EC00432=28.1117,15118.3294
EC00433=28.1001,15120.0000
EC00434=28.1117,15121.6706
EC00435=26.6025,15124.1349
EC00436=8.4383,15127.1678
EC00437=-0.0548,15127.9465
EC00438=-0.0188,15127.8844
EC00439=-0.0094,15127.7630
EC00440=-0.0057,15127.6803
EC00441=-0.5045,15127.7585
EC00442=-1.1939,15129.4604
EC00443=-0.7971,15132.4636
EC00444=-0.0543,15136.2505
EC00445=-0.0054,15140.3860
EC00446=-0.0052,15144.6140
EC00447=-0.0540,15148.7498
EC00448=-0.7993,15152.5363
EC00449=-1.1940,15155.5394
EC00450=-0.5081,15157.2413
EC00451=-0.0087,15157.3191
EC00452=-0.0113,15157.2369
EC00453=-0.0208,15157.1159
EC00454=-0.0563,15157.0536
EC00455=8.4405,15157.8325
EC00456=26.5997,15160.8660
EC00457=28.1098,15163.3290
EC00458=28.0967,15165.0000
EC00459=28.1098,15166.6710
EC00460=26.5997,15169.1340
EC00461=8.4405,15172.1675
EC00462=-0.0563,15172.9464
EC00463=-0.0208,15172.8841
EC00464=-0.0113,15172.7631
EC00465=-0.0087,15172.6809
EC00466=-0.5081,15172.7587
EC00467=-1.1940,15174.4606
EC00468=-0.7993,15177.4637
EC00469=-0.0540,15181.2502
EC00470=-0.0052,15185.3860
EC00471=-0.0054,15189.6140
EC00472=-0.0543,15193.7495
EC00473=-0.7971,15197.5364
EC00474=-1.1939,15200.5396
EC00475=-0.5045,15202.2415
EC00476=-0.0057,15202.3197
EC00477=-0.0094,15202.2370
EC00478=-0.0188,15202.1156
EC00479=-0.0548,15202.0535
EC00480=8.4383,15202.8322
EC00481=26.6025,15205.8651
EC00482=28.1117,15208.3294
EC00483=28.1001,15210.0000
EC00484=26.2576,15210.0000
EC00485=26.2720,15211.6025
EC00486=24.7331,15214.0449
EC00487=7.3770,15217.0981
EC00488=-0.0435,15217.8538
EC00489=-0.0134,15217.7815
EC00490=-0.0020,15217.6711
EC00491=-0.0031,15217.6022
EC00492=-0.3615,15217.6844
EC00493=-0.8397,15219.3971
EC00494=-0.5442,15222.4165
EC00495=-0.0362,15226.2223
EC00496=-0.0054,15230.3773
EC00497=-0.0052,15234.6227
EC00498=-0.0384,15238.7775
EC00499=-0.5441,15242.5833
EC00500=-0.8412,15245.6027
EC00501=-0.3666,15247.3159
EC00502=-0.0016,15247.3980
EC00503=-0.0027,15247.3291
EC00504=-0.0129,15247.2193
EC00505=-0.0389,15247.1468
EC00506=7.3773,15247.9017
EC00507=24.7330,15250.9551
EC00508=26.2704,15253.3970
EC00509=26.2558,15255.0000
EC00510=26.2704,15256.6030
EC00511=24.7330,15259.0449
EC00512=7.3727,15262.0983
EC00513=-0.0389,15262.8532
EC00514=-0.0129,15262.7807
EC00515=-0.0027,15262.6709
EC00516=-0.0016,15262.6020
EC00517=-0.3666,15262.6841
EC00518=-0.8412,15264.3973
EC00519=-0.5441,15267.4167
EC00520=-0.0384,15271.2225
EC00521=-0.0052,15275.3773
EC00522=-0.0054,15279.6227
EC00523=-0.0362,15283.7777
EC00524=-0.5442,15287.5835
EC00525=-0.8397,15290.6029
EC00526=-0.3615,15292.3156
EC00527=-0.0031,15292.3978
EC00528=-0.0020,15292.3289
EC00529=-0.0134,15292.2185
EC00530=-0.0435,15292.1462
EC00531=7.3770,15292.9019
EC00532=24.7331,15295.9551
EC00533=26.2720,15298.3975
EC00534=26.2576,15300.0000
EC00535=26.2720,15301.6025
EC00536=24.7327,15304.0449
EC00537=7.3770,15307.0981
EC00538=-0.0435,15307.8538
EC00539=-0.0134,15307.7815
EC00540=-0.0020,15307.6711
EC00541=-0.0031,15307.6022
EC00542=-0.3615,15307.6844
EC00543=-0.8397,15309.3971
EC00544=-0.5442,15312.4165
EC00545=-0.0362,15316.2223
EC00546=-0.0054,15320.3773
EC00547=-0.0052,15324.6227
EC00548=-0.0384,15328.7775
EC00549=-0.5441,15332.5833
EC00550=-0.8412,15335.6027
EC00551=-0.3666,15337.3159
EC00552=-0.0016,15337.3980
EC00553=-0.0027,15337.3291
EC00554=-0.0129,15337.2193
EC00555=-0.0389,15337.1468
EC00556=7.3773,15337.9017
EC00557=24.7330,15340.9551
EC00558=26.2704,15343.3970
EC00559=26.2558,15345.0000
EC00560=26.2704,15346.6030
EC00561=24.7330,15349.0449
EC00562=7.3727,15352.0983
EC00563=-0.0389,15352.8532
EC00564=-0.0129,15352.7807
EC00565=-0.0027,15352.6709
EC00566=-0.0016,15352.6020
EC00567=-0.3666,15352.6841
EC00568=-0.8412,15354.3973
EC00569=-0.5441,15357.4167
EC00570=-0.0384,15361.2225
EC00571=-0.0052,15365.3773
EC00572=-0.0054,15369.6227
EC00573=-0.0362,15373.7777
EC00574=-0.5442,15377.5835
EC00575=-0.8397,15380.6029
EC00576=-0.3615,15382.3156
EC00577=-0.0031,15382.3978
EC00578=-0.0020,15382.3289
EC00579=-0.0134,15382.2185
EC00580=-0.0435,15382.1462
EC00581=7.3770,15382.9019
EC00582=24.7331,15385.9551
EC00583=26.2720,15388.3975
EC00584=26.2576,15390.0000
EC00585=26.2576,15390.0000
EC00586=26.2720,15391.6025
EC00587=24.7327,15394.0449
EC00588=7.3770,15397.0981
EC00589=-0.0435,15397.8538
EC00590=-0.0134,15397.7815
EC00591=-0.0020,15397.6711
EC00592=-0.0031,15397.6022
EC00593=-0.3615,15397.6844
EC00594=-0.8397,15399.3971
EC00595=-0.5442,15402.4165
EC00596=-0.0362,15406.2223
EC00597=-0.0054,15410.3773
EC00598=-0.0052,15414.6227
EC00599=-0.0384,15418.7775
EC00600=-0.5441,15422.5833
EC00601=-0.8412,15425.6027
EC00602=-0.3666,15427.3159
EC00603=-0.0016,15427.3980
EC00604=-0.0027,15427.3291
EC00605=-0.0129,15427.2193
EC00606=-0.0389,15427.1468
EC00607=7.3773,15427.9017
EC00608=24.7330,15430.9551
EC00609=26.2704,15433.3970
EC00610=26.2558,15435.0000
EC00611=26.2704,15436.6030
EC00612=24.7330,15439.0449
EC00613=7.3727,15442.0983
EC00614=-0.0389,15442.8532
EC00615=-0.0129,15442.7807
EC00616=-0.0027,15442.6709
EC00617=-0.0016,15442.6020
EC00618=-0.3666,15442.6841
EC00619=-0.8412,15444.3973
EC00620=-0.5441,15447.4167
EC00621=-0.0384,15451.2225
EC00622=-0.0052,15455.3773
EC00623=-0.0054,15459.6227
EC00624=-0.0362,15463.7777
EC00625=-0.5442,15467.5835
EC00626=-0.8397,15470.6029
EC00627=-0.3615,15472.3156
EC00628=-0.0031,15472.3978
EC00629=-0.0020,15472.3289
EC00630=-0.0134,15472.2185
EC00631=-0.0435,15472.1462
EC00632=7.3770,15472.9019
EC00633=24.7331,15475.9551
EC00634=26.2720,15478.3975
EC00635=26.2576,15480.0000
EC00636=26.2720,15481.6025
EC00637=24.7327,15484.0449
EC00638=7.3770,15487.0981
EC00639=-0.0435,15487.8538
EC00640=-0.0134,15487.7815
EC00641=-0.0020,15487.6711
EC00642=-0.0031,15487.6022
EC00643=-0.3615,15487.6844
EC00644=-0.8397,15489.3971
EC00645=-0.5442,15492.4165
EC00646=-0.0362,15496.2223
EC00647=-0.0054,15500.3773
EC00648=-0.0052,15504.6227
EC00649=-0.0384,15508.7775
EC00650=-0.5441,15512.5833
EC00651=-0.8412,15515.6027
EC00652=-0.3666,15517.3159
EC00653=-0.0016,15517.3980
EC00654=-0.0027,15517.3291
EC00655=-0.0129,15517.2193
EC00656=-0.0389,15517.1468
EC00657=7.3773,15517.9017
EC00658=24.7330,15520.9551
EC00659=26.2704,15523.3970
EC00660=26.2558,15525.0000
EC00661=26.2704,15526.6030
EC00662=24.7330,15529.0449
EC00663=7.3727,15532.0983
EC00664=-0.0389,15532.8532
EC00665=-0.0129,15532.7807
EC00666=-0.0027,15532.6709
EC00667=-0.0016,15532.6020
EC00668=-0.3666,15532.6841
EC00669=-0.8412,15534.3973
EC00670=-0.5441,15537.4167
EC00671=-0.0384,15541.2225
EC00672=-0.0052,15545.3773
EC00673=-0.0054,15549.6227
EC00674=-0.0362,15553.7777
EC00675=-0.5442,15557.5835
EC00676=-0.8397,15560.6029
EC00677=-0.3615,15562.3156
EC00678=-0.0031,15562.3978
EC00679=-0.0020,15562.3289
EC00680=-0.0134,15562.2185
EC00681=-0.0435,15562.1462
EC00682=7.3770,15562.9019
EC00683=24.7327,15565.9551
EC00684=26.2720,15568.3975
EC00685=26.2576,15570.0000
EC00686=24.1993,15570.0000
EC00687=24.2117,15571.5376
EC00688=22.6760,15573.9586
EC00689=6.3608,15577.0327
EC00690=-0.0296,15577.7683
EC00691=-0.0072,15577.6919
EC00692=0.0012,15577.5966
EC00693=0.0004,15577.5446
EC00694=-0.2180,15577.6343
EC00695=-0.4664,15579.3569
EC00696=-0.2743,15582.3884
EC00697=-0.0181,15586.2065
EC00698=-0.0000,15590.3718
EC00699=-0.0000,15594.6278
EC00700=-0.0128,15598.7938
EC00701=-0.2776,15602.6119
EC00702=-0.4673,15605.6434
EC00703=-0.2176,15607.3659
EC00704=0.0009,15607.4553
EC00705=-0.0015,15607.4027
EC00706=-0.0071,15607.3085
EC00707=-0.0275,15607.2322
EC00708=6.3616,15607.9674
EC00709=22.6775,15611.0417
EC00710=24.2122,15613.4634
EC00711=24.1961,15615.0000
EC00712=24.2160,15616.5366
EC00713=22.6769,15618.9583
EC00714=6.3616,15622.0326
EC00715=-0.0275,15622.7678
EC00716=-0.0071,15622.6915
EC00717=-0.0015,15622.5973
EC00718=0.0009,15622.5447
EC00719=-0.2176,15622.6341
EC00720=-0.4673,15624.3566
EC00721=-0.2776,15627.3881
EC00722=-0.0128,15631.2062
EC00723=-0.0000,15635.3722
EC00724=-0.0000,15639.6282
EC00725=-0.0181,15643.7935
EC00726=-0.2743,15647.6116
EC00727=-0.4664,15650.6431
EC00728=-0.2180,15652.3657
EC00729=0.0004,15652.4554
EC00730=0.0012,15652.4034
EC00731=-0.0072,15652.3081
EC00732=-0.0296,15652.2317
EC00733=6.3608,15652.9673
EC00734=22.6760,15656.0414
EC00735=24.2117,15658.4624
EC00736=24.1993,15660.0000
EC00737=24.2117,15661.5365
EC00738=22.6760,15663.9586
EC00739=6.3608,15667.0327
EC00740=-0.0296,15667.7683
EC00741=-0.0072,15667.6919
EC00742=0.0012,15667.5966
EC00743=0.0004,15667.5446
EC00744=-0.2180,15667.6343
EC00745=-0.4664,15669.3569
EC00746=-0.2743,15672.3884
EC00747=-0.0181,15676.2065
EC00748=-0.0000,15680.3718
EC00749=-0.0000,15684.6278
EC00750=-0.0128,15688.7938
EC00751=-0.2776,15692.6119
EC00752=-0.4673,15695.6434
EC00753=-0.2176,15697.3659
EC00754=0.0009,15697.4553
EC00755=-0.0015,15697.4027
EC00756=-0.0071,15697.3085
EC00757=-0.0275,15697.2322
EC00758=6.3616,15697.9674
EC00759=22.6775,15701.0417
EC00760=24.2122,15703.4634
EC00761=24.1961,15705.0000
EC00762=24.2160,15706.5366
EC00763=22.6769,15708.9583
EC00764=6.3616,15712.0326
EC00765=-0.0275,15712.7678
EC00766=-0.0071,15712.6915
EC00767=-0.0015,15712.5973
EC00768=0.0009,15712.5447
EC00769=-0.2176,15712.6341
EC00770=-0.4673,15714.3566
EC00771=-0.2776,15717.3881
EC00772=-0.0128,15721.2062
EC00773=-0.0000,15725.3722
EC00774=-0.0000,15729.6282
EC00775=-0.0181,15733.7935
EC00776=-0.2743,15737.6116
EC00777=-0.4664,15740.6431
EC00778=-0.2180,15742.3657
EC00779=0.0004,15742.4554
EC00780=0.0012,15742.4034
EC00781=-0.0072,15742.3081
EC00782=-0.0296,15742.2317
EC00783=6.3608,15742.9673
EC00784=22.6760,15746.0414
EC00785=24.2117,15748.4624
EC00786=24.1993,15750.0000
EC00787=24.1993,15750.0000
EC00788=24.2117,15751.5365
EC00789=22.6760,15753.9586
EC00790=6.3608,15757.0327
EC00791=-0.0296,15757.7683
EC00792=-0.0072,15757.6919
EC00793=0.0012,15757.5966
EC00794=0.0004,15757.5446
EC00795=-0.2180,15757.6343
EC00796=-0.4664,15759.3569
EC00797=-0.2743,15762.3884
EC00798=-0.0181,15766.2065
EC00799=-0.0000,15770.3718
EC00800=-0.0000,15774.6278
EC00801=-0.0128,15778.7938
EC00802=-0.2776,15782.6119
EC00803=-0.4673,15785.6434
EC00804=-0.2176,15787.3659
EC00805=0.0009,15787.4553
EC00806=-0.0015,15787.4027
EC00807=-0.0071,15787.3085
EC00808=-0.0275,15787.2322
EC00809=6.3616,15787.9674
EC00810=22.6775,15791.0417
EC00811=24.2122,15793.4634
EC00812=24.1961,15795.0000
EC00813=24.2160,15796.5366
EC00814=22.6769,15798.9583
EC00815=6.3616,15802.0326
EC00816=-0.0275,15802.7678
EC00817=-0.0071,15802.6915
EC00818=-0.0015,15802.5973
EC00819=0.0009,15802.5447
EC00820=-0.2176,15802.6341
EC00821=-0.4673,15804.3566
EC00822=-0.2776,15807.3881
EC00823=-0.0128,15811.2062
EC00824=-0.0000,15815.3722
EC00825=-0.0000,15819.6282
EC00826=-0.0181,15823.7935
EC00827=-0.2743,15827.6116
EC00828=-0.4664,15830.6431
EC00829=-0.2180,15832.3657
EC00830=0.0004,15832.4554
EC00831=0.0012,15832.4034
EC00832=-0.0072,15832.3081
EC00833=-0.0296,15832.2317
EC00834=6.3608,15832.9673
EC00835=22.6760,15836.0414
EC00836=24.2117,15838.4624
EC00837=24.1993,15840.0000
EC00838=24.2117,15841.5365
EC00839=22.6760,15843.9586
EC00840=6.3608,15847.0327
EC00841=-0.0296,15847.7683
EC00842=-0.0072,15847.6919
EC00843=0.0012,15847.5966
EC00844=0.0004,15847.5446
EC00845=-0.2180,15847.6343
EC00846=-0.4664,15849.3569
EC00847=-0.2743,15852.3884
EC00848=-0.0181,15856.2065
EC00849=-0.0000,15860.3718
EC00850=-0.0000,15864.6278
EC00851=-0.0128,15868.7938
EC00852=-0.2776,15872.6119
EC00853=-0.4673,15875.6434
EC00854=-0.2176,15877.3659
EC00855=0.0009,15877.4553
EC00856=-0.0015,15877.4027
EC00857=-0.0071,15877.3085
EC00858=-0.0275,15877.2322
EC00859=6.3616,15877.9674
EC00860=22.6775,15881.0417
EC00861=24.2122,15883.4634
EC00862=24.1961,15885.0000
EC00863=24.2160,15886.5366
EC00864=22.6769,15888.9583
EC00865=6.3616,15892.0326
EC00866=-0.0275,15892.7678
EC00867=-0.0071,15892.6915
EC00868=-0.0015,15892.5973
EC00869=0.0009,15892.5447
EC00870=-0.2176,15892.6341
EC00871=-0.4673,15894.3566
EC00872=-0.2776,15897.3881
EC00873=-0.0128,15901.2062
EC00874=-0.0000,15905.3722
EC00875=-0.0000,15909.6282
EC00876=-0.0181,15913.7935
EC00877=-0.2743,15917.6116
EC00878=-0.4664,15920.6431
EC00879=-0.2180,15922.3657
EC00880=0.0004,15922.4554
EC00881=0.0012,15922.4034
EC00882=-0.0072,15922.3081
EC00883=-0.0296,15922.2317
EC00884=6.3608,15922.9673
EC00885=22.6760,15926.0414
EC00886=24.2117,15928.4635
EC00887=24.1993,15930.0000
EC00888=21.8993,15930.0000
EC00889=21.9171,15931.4747
EC00890=20.4142,15933.8756
EC00891=5.3944,15936.9699
EC00892=-0.0194,15937.6906
EC00893=-0.0061,15937.6170
EC00894=0.0006,15937.5429
EC00895=-0.0001,15937.5106
EC00896=-0.0677,15937.6094
EC00897=-0.0727,15939.3401
EC00898=-0.0715,15965.6602
EC00899=-0.0690,15967.3910
EC00900=-0.0010,15967.4898
EC00901=-0.0010,15967.4572
EC00902=-0.0014,15967.3834
EC00903=-0.0171,15967.3085
EC00904=5.3944,15968.0296
EC00905=20.4131,15971.1238
EC00906=21.9192,15973.5256
EC00907=21.8955,15975.0000
EC00908=21.9192,15976.4744
EC00909=20.4131,15978.8762
EC00910=5.3909,15981.9704
EC00911=-0.0171,15982.6915
EC00912=-0.0014,15982.6166
EC00913=-0.0010,15982.5428
EC00914=-0.0010,15982.5102
EC00915=-0.0690,15982.6090
EC00916=-0.0715,15984.3398
EC00917=-0.0727,16010.6599
EC00918=-0.0677,16012.3906
EC00919=-0.0001,16012.4894
EC00920=0.0006,16012.4571
EC00921=-0.0061,16012.3830
EC00922=-0.0194,16012.3094
EC00923=5.3944,16013.0301
EC00924=20.4142,16016.1244
EC00925=21.9171,16018.5253
EC00926=21.8993,16020.0000
EC00927=21.9171,16021.4736
EC00928=20.4141,16023.8767
EC00929=5.3944,16026.9699
EC00930=-0.0194,16027.6906
EC00931=-0.0061,16027.6170
EC00932=0.0006,16027.5429
EC00933=-0.0001,16027.5106
EC00934=-0.0677,16027.6094
EC00935=-0.0727,16029.3401
EC00936=-0.0715,16055.6602
EC00937=-0.0690,16057.3910
EC00938=-0.0010,16057.4898
EC00939=-0.0010,16057.4572
EC00940=-0.0014,16057.3834
EC00941=-0.0171,16057.3085
EC00942=5.3944,16058.0296
EC00943=20.4131,16061.1238
EC00944=21.9192,16063.5256
EC00945=21.8955,16065.0000
EC00946=21.9192,16066.4744
EC00947=20.4131,16068.8762
EC00948=5.3909,16071.9704
EC00949=-0.0171,16072.6915
EC00950=-0.0014,16072.6166
EC00951=-0.0010,16072.5428
EC00952=-0.0010,16072.5102
EC00953=-0.0690,16072.6090
EC00954=-0.0715,16074.3398
EC00955=-0.0727,16100.6599
EC00956=-0.0677,16102.3906
EC00957=-0.0001,16102.4894
EC00958=0.0006,16102.4571
EC00959=-0.0061,16102.3830
EC00960=-0.0194,16102.3094
EC00961=5.3944,16103.0301
EC00962=20.4142,16106.1244
EC00963=21.9171,16108.5253
EC00964=21.8993,16110.0000
EC00965=21.8993,16110.0000
EC00966=21.9171,16111.4736
EC00967=20.4141,16113.8767
EC00968=5.3944,16116.9699
EC00969=-0.0194,16117.6906
EC00970=-0.0061,16117.6170
EC00971=0.0006,16117.5429
EC00972=-0.0001,16117.5106
EC00973=-0.0677,16117.6094
EC00974=-0.0727,16119.3401
EC00975=-0.0715,16145.6602
EC00976=-0.0690,16147.3910
EC00977=-0.0010,16147.4898
EC00978=-0.0010,16147.4572
EC00979=-0.0014,16147.3834
EC00980=-0.0171,16147.3085
EC00981=5.3944,16148.0296
EC00982=20.4131,16151.1238
EC00983=21.9192,16153.5256
EC00984=21.8955,16155.0000
EC00985=21.9192,16156.4744
EC00986=20.4131,16158.8762
EC00987=5.3909,16161.9704
EC00988=-0.0171,16162.6915
EC00989=-0.0014,16162.6166
EC00990=-0.0010,16162.5428
EC00991=-0.0010,16162.5102
EC00992=-0.0690,16162.6090
EC00993=-0.0715,16164.3398
EC00994=-0.0727,16190.6599
EC00995=-0.0677,16192.3906
EC00996=-0.0001,16192.4894
EC00997=0.0006,16192.4571
EC00998=-0.0061,16192.3830
EC00999=-0.0194,16192.3094
EC01000=5.3944,16193.0301
EC01001=20.4142,16196.1244
EC01002=21.9171,16198.5253
EC01003=21.8993,16200.0000
EC01004=21.9171,16201.4736
EC01005=20.4141,16203.8767
EC01006=5.3944,16206.9699
EC01007=-0.0194,16207.6906
EC01008=-0.0061,16207.6170
EC01009=0.0006,16207.5429
EC01010=-0.0001,16207.5106
EC01011=-0.0677,16207.6094
EC01012=-0.0727,16209.3401
EC01013=-0.0715,16235.6602
EC01014=-0.0690,16237.3910
EC01015=-0.0010,16237.4898
EC01016=-0.0010,16237.4572
EC01017=-0.0014,16237.3834
EC01018=-0.0171,16237.3085
EC01019=5.3944,16238.0296
EC01020=20.4131,16241.1238
EC01021=21.9192,16243.5256
EC01022=21.8955,16245.0000
EC01023=21.9192,16246.4744
EC01024=20.4131,16248.8762
EC01025=5.3909,16251.9704
EC01026=-0.0171,16252.6915
EC01027=-0.0014,16252.6166
EC01028=-0.0010,16252.5428
EC01029=-0.0010,16252.5102
EC01030=-0.0690,16252.6090
EC01031=-0.0715,16254.3398
EC01032=-0.0727,16280.6599
EC01033=-0.0677,16282.3906
EC01034=-0.0001,16282.4894
EC01035=0.0006,16282.4571
EC01036=-0.0061,16282.3830
EC01037=-0.0194,16282.3094
EC01038=5.3944,16283.0301
EC01039=20.4141,16286.1233
EC01040=21.9171,16288.5264
EC01041=21.8993,16290.0000
EC01042=19.3355,16290.0000
EC01043=19.3601,16291.4165
EC01044=17.9316,16293.7994
EC01045=4.4629,16296.9134
EC01046=-0.0109,16297.6249
EC01047=-0.0035,16297.5584
EC01048=0.0012,16297.5104
EC01049=-0.0008,16327.4901
EC01050=-0.0004,16327.4412
EC01051=-0.0099,16327.3752
EC01052=4.4644,16328.0867
EC01053=17.9314,16331.2006
EC01054=19.3612,16333.5844
EC01055=19.3375,16335.0000
EC01056=19.3612,16336.4156
EC01057=17.9313,16338.8001
EC01058=4.4644,16341.9133
EC01059=-0.0099,16342.6248
EC01060=-0.0004,16342.5588
EC01061=-0.0008,16342.5099
EC01062=0.0012,16372.4896
EC01063=-0.0035,16372.4416
EC01064=-0.0109,16372.3751
EC01065=4.4629,16373.0866
EC01066=17.9316,16376.2006
EC01067=19.3601,16378.5835
EC01068=19.3355,16380.0000
EC01069=19.3601,16381.4153
EC01070=17.9315,16383.8005
EC01071=4.4629,16386.9134
EC01072=-0.0109,16387.6249
EC01073=-0.0035,16387.5584
EC01074=0.0012,16387.5104
EC01075=-0.0008,16417.4901
EC01076=-0.0004,16417.4412
EC01077=-0.0099,16417.3752
EC01078=4.4644,16418.0867
EC01079=17.9314,16421.2006
EC01080=19.3612,16423.5844
EC01081=19.3375,16425.0000
EC01082=19.3612,16426.4156
EC01083=17.9313,16428.8001
EC01084=4.4644,16431.9133
EC01085=-0.0099,16432.6248
EC01086=-0.0004,16432.5588
EC01087=-0.0008,16432.5099
EC01088=0.0012,16462.4896
EC01089=-0.0035,16462.4416
EC01090=-0.0109,16462.3751
EC01091=4.4629,16463.0866
EC01092=17.9316,16466.2006
EC01093=19.3601,16468.5835
EC01094=19.3355,16470.0000
EC01095=19.3355,16470.0000
EC01096=19.3601,16471.4153
EC01097=17.9315,16473.8005
EC01098=4.4629,16476.9134
EC01099=-0.0109,16477.6249
EC01100=-0.0035,16477.5584
EC01101=0.0012,16477.5104
EC01102=-0.0008,16507.4901
EC01103=-0.0004,16507.4412
EC01104=-0.0099,16507.3752
EC01105=4.4644,16508.0867
EC01106=17.9314,16511.2006
EC01107=19.3612,16513.5844
EC01108=19.3375,16515.0000
EC01109=19.3612,16516.4156
EC01110=17.9313,16518.8001
EC01111=4.4644,16521.9133
EC01112=-0.0099,16522.6248
EC01113=-0.0004,16522.5588
EC01114=-0.0008,16522.5099
EC01115=0.0012,16552.4896
EC01116=-0.0035,16552.4416
EC01117=-0.0109,16552.3751
EC01118=4.4629,16553.0866
EC01119=17.9316,16556.2006
EC01120=19.3601,16558.5835
EC01121=19.3355,16560.0000
EC01122=19.3601,16561.4153
EC01123=17.9315,16563.8005
EC01124=4.4629,16566.9134
EC01125=-0.0109,16567.6249
EC01126=-0.0035,16567.5584
EC01127=0.0012,16567.5104
EC01128=-0.0008,16597.4901
EC01129=-0.0004,16597.4412
EC01130=-0.0099,16597.3752
EC01131=4.4644,16598.0867
EC01132=17.9314,16601.2006
EC01133=19.3612,16603.5844
EC01134=19.3375,16605.0000
EC01135=19.3612,16606.4156
EC01136=17.9313,16608.8001
EC01137=4.4644,16611.9133
EC01138=-0.0099,16612.6248
EC01139=-0.0004,16612.5588
EC01140=-0.0008,16612.5099
EC01141=0.0012,16642.4896
EC01142=-0.0035,16642.4416
EC01143=-0.0109,16642.3751
EC01144=4.4629,16643.0866
EC01145=17.9315,16646.1995
EC01146=19.3601,16648.5847
EC01147=19.3355,16650.0000
EC01148=16.4995,16650.0000
EC01149=16.5281,16651.3641
EC01150=15.2268,16653.7307
EC01151=3.5661,16656.8641
EC01152=-0.0035,16657.5707
EC01153=0.0008,16657.5193
EC01154=0.0002,16687.4799
EC01155=-0.0013,16687.4296
EC01156=3.5658,16688.1360
EC01157=15.2245,16691.2692
EC01158=16.5280,16693.6362
EC01159=16.5019,16695.0000
EC01160=16.5280,16696.3630
EC01161=15.2245,16698.7308
EC01162=3.5623,16701.8640
EC01163=-0.0013,16702.5704
EC01164=0.0002,16702.5201
EC01165=0.0008,16732.4807
EC01166=-0.0035,16732.4293
EC01167=3.5661,16733.1359
EC01168=15.2268,16736.2693
EC01169=16.5281,16738.6359
EC01170=16.4995,16740.0000
EC01171=16.5281,16741.3630
EC01172=15.2212,16743.7318
EC01173=3.5661,16746.8641
EC01174=-0.0035,16747.5707
EC01175=0.0008,16747.5193
EC01176=0.0002,16777.4799
EC01177=-0.0013,16777.4296
EC01178=3.5658,16778.1360
EC01179=15.2245,16781.2692
EC01180=16.5280,16783.6362
EC01181=16.5019,16785.0000
EC01182=16.5280,16786.3630
EC01183=15.2245,16788.7308
EC01184=3.5623,16791.8640
EC01185=-0.0013,16792.5704
EC01186=0.0002,16792.5201
EC01187=0.0008,16822.4807
EC01188=-0.0035,16822.4293
EC01189=3.5661,16823.1359
EC01190=15.2268,16826.2693
EC01191=16.5281,16828.6359
EC01192=16.4995,16830.0000
EC01193=16.4995,16830.0000
EC01194=16.5281,16831.3630
EC01195=15.2212,16833.7318
EC01196=3.5661,16836.8641
EC01197=-0.0035,16837.5707
EC01198=0.0008,16837.5193
EC01199=0.0002,16867.4799
EC01200=-0.0013,16867.4296
EC01201=3.5658,16868.1360
EC01202=15.2245,16871.2692
EC01203=16.5280,16873.6362
EC01204=16.5019,16875.0000
EC01205=16.5280,16876.3630
EC01206=15.2245,16878.7308
EC01207=3.5623,16881.8640
EC01208=-0.0013,16882.5704
EC01209=0.0002,16882.5201
EC01210=0.0008,16912.4807
EC01211=-0.0035,16912.4293
EC01212=3.5661,16913.1359
EC01213=15.2268,16916.2693
EC01214=16.5281,16918.6359
EC01215=16.4995,16920.0000
EC01216=16.5281,16921.3630
EC01217=15.2212,16923.7318
EC01218=3.5661,16926.8641
EC01219=-0.0035,16927.5707
EC01220=0.0008,16927.5193
EC01221=0.0002,16957.4799
EC01222=-0.0013,16957.4296
EC01223=3.5658,16958.1360
EC01224=15.2245,16961.2692
EC01225=16.5280,16963.6362
EC01226=16.5019,16965.0000
EC01227=16.5280,16966.3630
EC01228=15.2245,16968.7308
EC01229=3.5623,16971.8640
EC01230=-0.0013,16972.5704
EC01231=0.0002,16972.5201
EC01232=0.0008,17002.4807
EC01233=-0.0035,17002.4293
EC01234=3.5661,17003.1359
EC01235=15.2212,17006.2682
EC01236=16.5281,17008.6370
EC01237=16.4995,17010.0000
EC01238=13.3790,17010.0000
EC01239=13.4131,17011.3191
EC01240=12.2840,17013.6720
EC01241=2.6850,17016.8225
EC01242=-0.0028,17017.5303
EC01243=0.0000,17017.5014
EC01244=0.0010,17047.4983
EC01245=0.0007,17047.4688
EC01246=2.6894,17048.1772
EC01247=12.2833,17051.3279
EC01248=13.4108,17053.6816
EC01249=13.3770,17055.0000
EC01250=13.4108,17056.3184
EC01251=12.2833,17058.6728
EC01252=2.6858,17061.8228
EC01253=0.0007,17062.5312
EC01254=0.0010,17062.5017
EC01255=0.0000,17092.4986
EC01256=-0.0028,17092.4697
EC01257=2.6850,17093.1775
EC01258=12.2840,17096.3280
EC01259=13.4131,17098.6809
EC01260=13.3790,17100.0000
EC01261=13.4131,17101.3180
EC01262=12.2840,17103.6719
EC01263=2.6850,17106.8225
EC01264=-0.0028,17107.5303
EC01265=0.0000,17107.5014
EC01266=0.0010,17137.4983
EC01267=0.0007,17137.4688
EC01268=2.6894,17138.1772
EC01269=12.2833,17141.3279
EC01270=13.4108,17143.6816
EC01271=13.3770,17145.0000
EC01272=13.4108,17146.3184
EC01273=12.2833,17148.6728
EC01274=2.6858,17151.8228
EC01275=0.0007,17152.5312
EC01276=0.0010,17152.5017
EC01277=0.0000,17182.4986
EC01278=-0.0028,17182.4697
EC01279=2.6850,17183.1775
EC01280=12.2840,17186.3280
EC01281=13.4131,17188.6809
EC01282=13.3790,17190.0000
EC01283=13.3790,17190.0000
EC01284=13.4131,17191.3180
EC01285=12.2840,17193.6719
EC01286=2.6850,17196.8225
EC01287=-0.0028,17197.5303
EC01288=0.0000,17197.5014
EC01289=0.0010,17227.4983
EC01290=0.0007,17227.4688
EC01291=2.6894,17228.1772
EC01292=12.2833,17231.3279
EC01293=13.4108,17233.6816
EC01294=13.3770,17235.0000
EC01295=13.4108,17236.3184
EC01296=12.2833,17238.6728
EC01297=2.6858,17241.8228
EC01298=0.0007,17242.5312
EC01299=0.0010,17242.5017
EC01300=0.0000,17272.4986
EC01301=-0.0028,17272.4697
EC01302=2.6850,17273.1775
EC01303=12.2840,17276.3280
EC01304=13.4131,17278.6809
EC01305=13.3790,17280.0000
EC01306=13.4131,17281.3180
EC01307=12.2840,17283.6719
EC01308=2.6850,17286.8225
EC01309=-0.0028,17287.5303
EC01310=0.0000,17287.5014
EC01311=0.0010,17317.4983
EC01312=0.0007,17317.4688
EC01313=2.6894,17318.1772
EC01314=12.2833,17321.3279
EC01315=13.4108,17323.6816
EC01316=13.3770,17325.0000
EC01317=13.4108,17326.3184
EC01318=12.2833,17328.6728
EC01319=2.6858,17331.8228
EC01320=0.0007,17332.5312
EC01321=0.0010,17332.5017
EC01322=0.0000,17362.4986
EC01323=-0.0028,17362.4697
EC01324=2.6850,17363.1775
EC01325=12.2840,17366.3281
EC01326=13.4131,17368.6820
EC01327=13.3790,17370.0000
EC01328=9.9625,17370.0000
EC01329=10.0055,17371.2828
EC01330=9.1102,17373.6251
EC01331=1.8184,17376.7919
EC01332=-0.0002,17377.5071
EC01333=-0.0019,17407.4934
EC01334=1.8180,17408.2087
EC01335=9.1088,17411.3754
EC01336=10.0034,17413.7178
EC01337=9.9681,17415.0000
EC01338=10.0034,17416.2813
EC01339=9.1045,17418.6253
EC01340=1.8180,17421.7913
EC01341=-0.0019,17422.5066
EC01342=-0.0002,17452.4929
EC01343=1.8184,17453.2081
EC01344=9.1102,17456.3749
EC01345=10.0055,17458.7172
EC01346=9.9625,17460.0000
EC01347=10.0055,17461.2817
EC01348=9.1102,17463.6251
EC01349=1.8184,17466.7919
EC01350=-0.0002,17467.5071
EC01351=-0.0019,17497.4934
EC01352=1.8180,17498.2087
EC01353=9.1088,17501.3754
EC01354=10.0034,17503.7178
EC01355=9.9681,17505.0000
EC01356=10.0034,17506.2813
EC01357=9.1045,17508.6253
EC01358=1.8180,17511.7913
EC01359=-0.0019,17512.5066
EC01360=-0.0002,17542.4929
EC01361=1.8184,17543.2081
EC01362=9.1102,17546.3749
EC01363=10.0055,17548.7172
EC01364=9.9625,17550.0000
EC01365=9.9625,17550.0000
EC01366=10.0055,17551.2817
EC01367=9.1102,17553.6251
EC01368=1.8184,17556.7919
EC01369=-0.0002,17557.5071
EC01370=-0.0019,17587.4934
EC01371=1.8180,17588.2087
EC01372=9.1088,17591.3754
EC01373=10.0034,17593.7178
EC01374=9.9681,17595.0000
EC01375=10.0034,17596.2813
EC01376=9.1045,17598.6253
EC01377=1.8180,17601.7913
EC01378=-0.0019,17602.5066
EC01379=-0.0002,17632.4929
EC01380=1.8184,17633.2081
EC01381=9.1102,17636.3749
EC01382=10.0055,17638.7172
EC01383=9.9625,17640.0000
EC01384=10.0055,17641.2817
EC01385=9.1102,17643.6251
EC01386=1.8184,17646.7919
EC01387=-0.0002,17647.5071
EC01388=-0.0019,17677.4934
EC01389=1.8180,17678.2087
EC01390=9.1088,17681.3754
EC01391=10.0034,17683.7178
EC01392=9.9681,17685.0000
EC01393=10.0034,17686.2813
EC01394=9.1045,17688.6253
EC01395=1.8180,17691.7913
EC01396=-0.0019,17692.5066
EC01397=-0.0002,17722.4929
EC01398=1.8184,17723.2081
EC01399=9.1102,17726.3749
EC01400=10.0055,17728.7183
EC01401=9.9625,17730.0000
EC01402=6.2750,17730.0000
EC01403=6.3226,17731.2567
EC01404=5.7076,17733.5913
EC01405=0.9490,17736.7714
EC01406=0.9504,17768.2287
EC01407=5.7094,17771.4086
EC01408=6.3224,17773.7431
EC01409=6.2761,17775.0000
EC01410=6.3224,17776.2560
EC01411=5.7094,17778.5914
EC01412=0.9504,17781.7713
EC01413=0.9490,17813.2286
EC01414=5.7076,17816.4087
EC01415=6.3226,17818.7433
EC01416=6.2750,17820.0000
EC01417=6.3226,17821.2567
EC01418=5.7073,17823.5913
EC01419=0.9490,17826.7713
EC01420=0.9504,17858.2287
EC01421=5.7094,17861.4086
EC01422=6.3224,17863.7431
EC01423=6.2761,17865.0000
EC01424=6.3224,17866.2560
EC01425=5.7094,17868.5914
EC01426=0.9504,17871.7713
EC01427=0.9490,17903.2286
EC01428=5.7076,17906.4087
EC01429=6.3226,17908.7433
EC01430=6.2750,17910.0000
EC01431=6.2750,17910.0000
EC01432=6.3226,17911.2567
EC01433=5.7073,17913.5913
EC01434=0.9490,17916.7713
EC01435=0.9504,17948.2287
EC01436=5.7094,17951.4086
EC01437=6.3224,17953.7431
EC01438=6.2761,17955.0000
EC01439=6.3224,17956.2560
EC01440=5.7094,17958.5914
EC01441=0.9504,17961.7713
EC01442=0.9490,17993.2286
EC01443=5.7076,17996.4087
EC01444=6.3226,17998.7433
EC01445=6.2750,18000.0000
EC01446=6.3226,18001.2567
EC01447=5.7073,18003.5913
EC01448=0.9490,18006.7713
EC01449=0.9504,18038.2287
EC01450=5.7094,18041.4086
EC01451=6.3224,18043.7431
EC01452=6.2761,18045.0000
EC01453=6.3224,18046.2560
EC01454=5.7094,18048.5914
EC01455=0.9504,18051.7713
EC01456=0.9490,18083.2287
EC01457=5.7073,18086.4087
EC01458=6.3226,18088.7433
EC01459=6.2750,18090.0000
EC01460=2.3325,18090.0000
EC01461=2.3906,18091.2432
EC01462=2.1024,18093.5737
EC01463=0.0582,18096.7645
EC01464=0.0539,18128.2351
EC01465=2.1022,18131.4267
EC01466=2.3916,18133.7573
EC01467=2.3342,18135.0000
EC01468=2.3916,18136.2427
EC01469=2.1022,18138.5742
EC01470=0.0539,18141.7649
EC01471=0.0582,18173.2355
EC01472=2.1024,18176.4263
EC01473=2.3906,18178.7568
EC01474=2.3325,18180.0000
EC01475=2.3906,18181.2420
EC01476=2.1024,18183.5737
EC01477=0.0582,18186.7645
EC01478=0.0539,18218.2351
EC01479=2.1022,18221.4267
EC01480=2.3916,18223.7573
EC01481=2.3342,18225.0000
EC01482=2.3916,18226.2427
EC01483=2.1022,18228.5742
EC01484=0.0539,18231.7649
EC01485=0.0582,18263.2355
EC01486=2.1024,18266.4263
EC01487=2.3906,18268.7568
EC01488=2.3325,18270.0000
EC01489=2.3325,18270.0000
EC01490=2.3906,18271.2420
EC01491=2.1024,18273.5737
EC01492=0.0582,18276.7645
EC01493=0.0539,18308.2351
EC01494=2.1022,18311.4267
EC01495=2.3916,18313.7573
EC01496=2.3342,18315.0000
EC01497=2.3916,18316.2427
EC01498=2.1022,18318.5742
EC01499=0.0539,18321.7649
EC01500=0.0582,18353.2355
EC01501=2.1024,18356.4263
EC01502=2.3906,18358.7568
EC01503=2.3325,18360.0000
EC01504=2.3906,18361.2420
EC01505=2.1024,18363.5737
EC01506=0.0582,18366.7645
EC01507=0.0539,18398.2351
EC01508=2.1022,18401.4267
EC01509=2.3916,18403.7573
EC01510=2.3342,18405.0000
EC01511=2.3916,18406.2427
EC01512=2.1022,18408.5742
EC01513=0.0539,18411.7649
EC01514=0.0582,18443.2355
EC01515=2.1024,18446.4263
EC01516=2.3906,18448.7580
EC01517=2.3325,18450.0000
//INST
///DATE 2021/09/24 14:37
///COMM
///ATTR SC,RW,RJ
////FRAME USER 2
///GROUP1 RB1
///GROUP2 ST1
NOP
SMOVL C00000 +MOVJ EC00000
SMOVL C00001 +MOVJ EC00001
SMOVL C00002 +MOVJ EC00002
SMOVL C00003 +MOVJ EC00003
SMOVL C00004 +MOVJ EC00004
SMOVL C00005 +MOVJ EC00005
SMOVL C00006 +MOVJ EC00006
SMOVL C00007 +MOVJ EC00007
SMOVL C00008 +MOVJ EC00008
SMOVL C00009 +MOVJ EC00009
SMOVL C00010 +MOVJ EC00010
SMOVL C00011 +MOVJ EC00011
SMOVL C00012 +MOVJ EC00012
SMOVL C00013 +MOVJ EC00013
SMOVL C00014 +MOVJ EC00014
SMOVL C00015 +MOVJ EC00015
SMOVL C00016 +MOVJ EC00016
SMOVL C00017 +MOVJ EC00017
SMOVL C00018 +MOVJ EC00018
SMOVL C00019 +MOVJ EC00019
SMOVL C00020 +MOVJ EC00020
SMOVL C00021 +MOVJ EC00021
SMOVL C00022 +MOVJ EC00022
SMOVL C00023 +MOVJ EC00023
SMOVL C00024 +MOVJ EC00024
SMOVL C00025 +MOVJ EC00025
SMOVL C00026 +MOVJ EC00026
SMOVL C00027 +MOVJ EC00027
SMOVL C00028 +MOVJ EC00028
SMOVL C00029 +MOVJ EC00029
SMOVL C00030 +MOVJ EC00030
SMOVL C00031 +MOVJ EC00031
SMOVL C00032 +MOVJ EC00032
SMOVL C00033 +MOVJ EC00033
SMOVL C00034 +MOVJ EC00034
SMOVL C00035 +MOVJ EC00035
SMOVL C00036 +MOVJ EC00036
SMOVL C00037 +MOVJ EC00037
SMOVL C00038 +MOVJ EC00038
SMOVL C00039 +MOVJ EC00039
SMOVL C00040 +MOVJ EC00040
SMOVL C00041 +MOVJ EC00041
SMOVL C00042 +MOVJ EC00042
SMOVL C00043 +MOVJ EC00043
SMOVL C00044 +MOVJ EC00044
SMOVL C00045 +MOVJ EC00045
SMOVL C00046 +MOVJ EC00046
SMOVL C00047 +MOVJ EC00047
SMOVL C00048 +MOVJ EC00048
SMOVL C00049 +MOVJ EC00049
SMOVL C00050 +MOVJ EC00050
SMOVL C00051 +MOVJ EC00051
SMOVL C00052 +MOVJ EC00052
SMOVL C00053 +MOVJ EC00053
SMOVL C00054 +MOVJ EC00054
SMOVL C00055 +MOVJ EC00055
SMOVL C00056 +MOVJ EC00056
SMOVL C00057 +MOVJ EC00057
SMOVL C00058 +MOVJ EC00058
SMOVL C00059 +MOVJ EC00059
SMOVL C00060 +MOVJ EC00060
SMOVL C00061 +MOVJ EC00061
SMOVL C00062 +MOVJ EC00062
SMOVL C00063 +MOVJ EC00063
SMOVL C00064 +MOVJ EC00064
SMOVL C00065 +MOVJ EC00065
SMOVL C00066 +MOVJ EC00066
SMOVL C00067 +MOVJ EC00067
SMOVL C00068 +MOVJ EC00068
SMOVL C00069 +MOVJ EC00069
SMOVL C00070 +MOVJ EC00070
SMOVL C00071 +MOVJ EC00071
SMOVL C00072 +MOVJ EC00072
SMOVL C00073 +MOVJ EC00073
SMOVL C00074 +MOVJ EC00074
SMOVL C00075 +MOVJ EC00075
SMOVL C00076 +MOVJ EC00076
SMOVL C00077 +MOVJ EC00077
SMOVL C00078 +MOVJ EC00078
SMOVL C00079 +MOVJ EC00079
SMOVL C00080 +MOVJ EC00080
SMOVL C00081 +MOVJ EC00081
SMOVL C00082 +MOVJ EC00082
SMOVL C00083 +MOVJ EC00083
SMOVL C00084 +MOVJ EC00084
SMOVL C00085 +MOVJ EC00085
SMOVL C00086 +MOVJ EC00086
SMOVL C00087 +MOVJ EC00087
SMOVL C00088 +MOVJ EC00088
SMOVL C00089 +MOVJ EC00089
SMOVL C00090 +MOVJ EC00090
SMOVL C00091 +MOVJ EC00091
SMOVL C00092 +MOVJ EC00092
SMOVL C00093 +MOVJ EC00093
SMOVL C00094 +MOVJ EC00094
SMOVL C00095 +MOVJ EC00095
SMOVL C00096 +MOVJ EC00096
SMOVL C00097 +MOVJ EC00097
SMOVL C00098 +MOVJ EC00098
SMOVL C00099 +MOVJ EC00099
SMOVL C00100 +MOVJ EC00100
SMOVL C00101 +MOVJ EC00101
SMOVL C00102 +MOVJ EC00102
SMOVL C00103 +MOVJ EC00103
SMOVL C00104 +MOVJ EC00104
SMOVL C00105 +MOVJ EC00105
SMOVL C00106 +MOVJ EC00106
SMOVL C00107 +MOVJ EC00107
SMOVL C00108 +MOVJ EC00108
SMOVL C00109 +MOVJ EC00109
SMOVL C00110 +MOVJ EC00110
SMOVL C00111 +MOVJ EC00111
SMOVL C00112 +MOVJ EC00112
SMOVL C00113 +MOVJ EC00113
SMOVL C00114 +MOVJ EC00114
SMOVL C00115 +MOVJ EC00115
SMOVL C00116 +MOVJ EC00116
SMOVL C00117 +MOVJ EC00117
SMOVL C00118 +MOVJ EC00118
SMOVL C00119 +MOVJ EC00119
SMOVL C00120 +MOVJ EC00120
SMOVL C00121 +MOVJ EC00121
SMOVL C00122 +MOVJ EC00122
SMOVL C00123 +MOVJ EC00123
SMOVL C00124 +MOVJ EC00124
SMOVL C00125 +MOVJ EC00125
SMOVL C00126 +MOVJ EC00126
SMOVL C00127 +MOVJ EC00127
SMOVL C00128 +MOVJ EC00128
SMOVL C00129 +MOVJ EC00129
SMOVL C00130 +MOVJ EC00130
SMOVL C00131 +MOVJ EC00131
SMOVL C00132 +MOVJ EC00132
SMOVL C00133 +MOVJ EC00133
SMOVL C00134 +MOVJ EC00134
SMOVL C00135 +MOVJ EC00135
SMOVL C00136 +MOVJ EC00136
SMOVL C00137 +MOVJ EC00137
SMOVL C00138 +MOVJ EC00138
SMOVL C00139 +MOVJ EC00139
SMOVL C00140 +MOVJ EC00140
SMOVL C00141 +MOVJ EC00141
SMOVL C00142 +MOVJ EC00142
SMOVL C00143 +MOVJ EC00143
SMOVL C00144 +MOVJ EC00144
SMOVL C00145 +MOVJ EC00145
SMOVL C00146 +MOVJ EC00146
SMOVL C00147 +MOVJ EC00147
SMOVL C00148 +MOVJ EC00148
SMOVL C00149 +MOVJ EC00149
SMOVL C00150 +MOVJ EC00150
SMOVL C00151 +MOVJ EC00151
SMOVL C00152 +MOVJ EC00152
SMOVL C00153 +MOVJ EC00153
SMOVL C00154 +MOVJ EC00154
SMOVL C00155 +MOVJ EC00155
SMOVL C00156 +MOVJ EC00156
SMOVL C00157 +MOVJ EC00157
SMOVL C00158 +MOVJ EC00158
SMOVL C00159 +MOVJ EC00159
SMOVL C00160 +MOVJ EC00160
SMOVL C00161 +MOVJ EC00161
SMOVL C00162 +MOVJ EC00162
SMOVL C00163 +MOVJ EC00163
SMOVL C00164 +MOVJ EC00164
SMOVL C00165 +MOVJ EC00165
SMOVL C00166 +MOVJ EC00166
SMOVL C00167 +MOVJ EC00167
SMOVL C00168 +MOVJ EC00168
SMOVL C00169 +MOVJ EC00169
SMOVL C00170 +MOVJ EC00170
SMOVL C00171 +MOVJ EC00171
SMOVL C00172 +MOVJ EC00172
SMOVL C00173 +MOVJ EC00173
SMOVL C00174 +MOVJ EC00174
SMOVL C00175 +MOVJ EC00175
SMOVL C00176 +MOVJ EC00176
SMOVL C00177 +MOVJ EC00177
SMOVL C00178 +MOVJ EC00178
SMOVL C00179 +MOVJ EC00179
SMOVL C00180 +MOVJ EC00180
SMOVL C00181 +MOVJ EC00181
SMOVL C00182 +MOVJ EC00182
SMOVL C00183 +MOVJ EC00183
SMOVL C00184 +MOVJ EC00184
SMOVL C00185 +MOVJ EC00185
SMOVL C00186 +MOVJ EC00186
SMOVL C00187 +MOVJ EC00187
SMOVL C00188 +MOVJ EC00188
SMOVL C00189 +MOVJ EC00189
SMOVL C00190 +MOVJ EC00190
SMOVL C00191 +MOVJ EC00191
SMOVL C00192 +MOVJ EC00192
SMOVL C00193 +MOVJ EC00193
SMOVL C00194 +MOVJ EC00194
SMOVL C00195 +MOVJ EC00195
SMOVL C00196 +MOVJ EC00196
SMOVL C00197 +MOVJ EC00197
SMOVL C00198 +MOVJ EC00198
SMOVL C00199 +MOVJ EC00199
SMOVL C00200 +MOVJ EC00200
SMOVL C00201 +MOVJ EC00201
SMOVL C00202 +MOVJ EC00202
SMOVL C00203 +MOVJ EC00203
SMOVL C00204 +MOVJ EC00204
SMOVL C00205 +MOVJ EC00205
SMOVL C00206 +MOVJ EC00206
SMOVL C00207 +MOVJ EC00207
SMOVL C00208 +MOVJ EC00208
SMOVL C00209 +MOVJ EC00209
SMOVL C00210 +MOVJ EC00210
SMOVL C00211 +MOVJ EC00211
SMOVL C00212 +MOVJ EC00212
SMOVL C00213 +MOVJ EC00213
SMOVL C00214 +MOVJ EC00214
SMOVL C00215 +MOVJ EC00215
SMOVL C00216 +MOVJ EC00216
SMOVL C00217 +MOVJ EC00217
SMOVL C00218 +MOVJ EC00218
SMOVL C00219 +MOVJ EC00219
SMOVL C00220 +MOVJ EC00220
SMOVL C00221 +MOVJ EC00221
SMOVL C00222 +MOVJ EC00222
SMOVL C00223 +MOVJ EC00223
SMOVL C00224 +MOVJ EC00224
SMOVL C00225 +MOVJ EC00225
SMOVL C00226 +MOVJ EC00226
SMOVL C00227 +MOVJ EC00227
SMOVL C00228 +MOVJ EC00228
SMOVL C00229 +MOVJ EC00229
SMOVL C00230 +MOVJ EC00230
SMOVL C00231 +MOVJ EC00231
SMOVL C00232 +MOVJ EC00232
SMOVL C00233 +MOVJ EC00233
SMOVL C00234 +MOVJ EC00234
SMOVL C00235 +MOVJ EC00235
SMOVL C00236 +MOVJ EC00236
SMOVL C00237 +MOVJ EC00237
SMOVL C00238 +MOVJ EC00238
SMOVL C00239 +MOVJ EC00239
SMOVL C00240 +MOVJ EC00240
SMOVL C00241 +MOVJ EC00241
SMOVL C00242 +MOVJ EC00242
SMOVL C00243 +MOVJ EC00243
SMOVL C00244 +MOVJ EC00244
SMOVL C00245 +MOVJ EC00245
SMOVL C00246 +MOVJ EC00246
SMOVL C00247 +MOVJ EC00247
SMOVL C00248 +MOVJ EC00248
SMOVL C00249 +MOVJ EC00249
SMOVL C00250 +MOVJ EC00250
SMOVL C00251 +MOVJ EC00251
SMOVL C00252 +MOVJ EC00252
SMOVL C00253 +MOVJ EC00253
SMOVL C00254 +MOVJ EC00254
SMOVL C00255 +MOVJ EC00255
SMOVL C00256 +MOVJ EC00256
SMOVL C00257 +MOVJ EC00257
SMOVL C00258 +MOVJ EC00258
SMOVL C00259 +MOVJ EC00259
SMOVL C00260 +MOVJ EC00260
SMOVL C00261 +MOVJ EC00261
SMOVL C00262 +MOVJ EC00262
SMOVL C00263 +MOVJ EC00263
SMOVL C00264 +MOVJ EC00264
SMOVL C00265 +MOVJ EC00265
SMOVL C00266 +MOVJ EC00266
SMOVL C00267 +MOVJ EC00267
SMOVL C00268 +MOVJ EC00268
SMOVL C00269 +MOVJ EC00269
SMOVL C00270 +MOVJ EC00270
SMOVL C00271 +MOVJ EC00271
SMOVL C00272 +MOVJ EC00272
SMOVL C00273 +MOVJ EC00273
SMOVL C00274 +MOVJ EC00274
SMOVL C00275 +MOVJ EC00275
SMOVL C00276 +MOVJ EC00276
SMOVL C00277 +MOVJ EC00277
SMOVL C00278 +MOVJ EC00278
SMOVL C00279 +MOVJ EC00279
SMOVL C00280 +MOVJ EC00280
SMOVL C00281 +MOVJ EC00281
SMOVL C00282 +MOVJ EC00282
SMOVL C00283 +MOVJ EC00283
SMOVL C00284 +MOVJ EC00284
SMOVL C00285 +MOVJ EC00285
SMOVL C00286 +MOVJ EC00286
SMOVL C00287 +MOVJ EC00287
SMOVL C00288 +MOVJ EC00288
SMOVL C00289 +MOVJ EC00289
SMOVL C00290 +MOVJ EC00290
SMOVL C00291 +MOVJ EC00291
SMOVL C00292 +MOVJ EC00292
SMOVL C00293 +MOVJ EC00293
SMOVL C00294 +MOVJ EC00294
SMOVL C00295 +MOVJ EC00295
SMOVL C00296 +MOVJ EC00296
SMOVL C00297 +MOVJ EC00297
SMOVL C00298 +MOVJ EC00298
SMOVL C00299 +MOVJ EC00299
SMOVL C00300 +MOVJ EC00300
SMOVL C00301 +MOVJ EC00301
SMOVL C00302 +MOVJ EC00302
SMOVL C00303 +MOVJ EC00303
SMOVL C00304 +MOVJ EC00304
SMOVL C00305 +MOVJ EC00305
SMOVL C00306 +MOVJ EC00306
SMOVL C00307 +MOVJ EC00307
SMOVL C00308 +MOVJ EC00308
SMOVL C00309 +MOVJ EC00309
SMOVL C00310 +MOVJ EC00310
SMOVL C00311 +MOVJ EC00311
SMOVL C00312 +MOVJ EC00312
SMOVL C00313 +MOVJ EC00313
SMOVL C00314 +MOVJ EC00314
SMOVL C00315 +MOVJ EC00315
SMOVL C00316 +MOVJ EC00316
SMOVL C00317 +MOVJ EC00317
SMOVL C00318 +MOVJ EC00318
SMOVL C00319 +MOVJ EC00319
SMOVL C00320 +MOVJ EC00320
SMOVL C00321 +MOVJ EC00321
SMOVL C00322 +MOVJ EC00322
SMOVL C00323 +MOVJ EC00323
SMOVL C00324 +MOVJ EC00324
SMOVL C00325 +MOVJ EC00325
SMOVL C00326 +MOVJ EC00326
SMOVL C00327 +MOVJ EC00327
SMOVL C00328 +MOVJ EC00328
SMOVL C00329 +MOVJ EC00329
SMOVL C00330 +MOVJ EC00330
SMOVL C00331 +MOVJ EC00331
SMOVL C00332 +MOVJ EC00332
SMOVL C00333 +MOVJ EC00333
SMOVL C00334 +MOVJ EC00334
SMOVL C00335 +MOVJ EC00335
SMOVL C00336 +MOVJ EC00336
SMOVL C00337 +MOVJ EC00337
SMOVL C00338 +MOVJ EC00338
SMOVL C00339 +MOVJ EC00339
SMOVL C00340 +MOVJ EC00340
SMOVL C00341 +MOVJ EC00341
SMOVL C00342 +MOVJ EC00342
SMOVL C00343 +MOVJ EC00343
SMOVL C00344 +MOVJ EC00344
SMOVL C00345 +MOVJ EC00345
SMOVL C00346 +MOVJ EC00346
SMOVL C00347 +MOVJ EC00347
SMOVL C00348 +MOVJ EC00348
SMOVL C00349 +MOVJ EC00349
SMOVL C00350 +MOVJ EC00350
SMOVL C00351 +MOVJ EC00351
SMOVL C00352 +MOVJ EC00352
SMOVL C00353 +MOVJ EC00353
SMOVL C00354 +MOVJ EC00354
SMOVL C00355 +MOVJ EC00355
SMOVL C00356 +MOVJ EC00356
SMOVL C00357 +MOVJ EC00357
SMOVL C00358 +MOVJ EC00358
SMOVL C00359 +MOVJ EC00359
SMOVL C00360 +MOVJ EC00360
SMOVL C00361 +MOVJ EC00361
SMOVL C00362 +MOVJ EC00362
SMOVL C00363 +MOVJ EC00363
SMOVL C00364 +MOVJ EC00364
SMOVL C00365 +MOVJ EC00365
SMOVL C00366 +MOVJ EC00366
SMOVL C00367 +MOVJ EC00367
SMOVL C00368 +MOVJ EC00368
SMOVL C00369 +MOVJ EC00369
SMOVL C00370 +MOVJ EC00370
SMOVL C00371 +MOVJ EC00371
SMOVL C00372 +MOVJ EC00372
SMOVL C00373 +MOVJ EC00373
SMOVL C00374 +MOVJ EC00374
SMOVL C00375 +MOVJ EC00375
SMOVL C00376 +MOVJ EC00376
SMOVL C00377 +MOVJ EC00377
SMOVL C00378 +MOVJ EC00378
SMOVL C00379 +MOVJ EC00379
SMOVL C00380 +MOVJ EC00380
SMOVL C00381 +MOVJ EC00381
SMOVL C00382 +MOVJ EC00382
SMOVL C00383 +MOVJ EC00383
SMOVL C00384 +MOVJ EC00384
SMOVL C00385 +MOVJ EC00385
SMOVL C00386 +MOVJ EC00386
SMOVL C00387 +MOVJ EC00387
SMOVL C00388 +MOVJ EC00388
SMOVL C00389 +MOVJ EC00389
SMOVL C00390 +MOVJ EC00390
SMOVL C00391 +MOVJ EC00391
SMOVL C00392 +MOVJ EC00392
SMOVL C00393 +MOVJ EC00393
SMOVL C00394 +MOVJ EC00394
SMOVL C00395 +MOVJ EC00395
SMOVL C00396 +MOVJ EC00396
SMOVL C00397 +MOVJ EC00397
SMOVL C00398 +MOVJ EC00398
SMOVL C00399 +MOVJ EC00399
SMOVL C00400 +MOVJ EC00400
SMOVL C00401 +MOVJ EC00401
SMOVL C00402 +MOVJ EC00402
SMOVL C00403 +MOVJ EC00403
SMOVL C00404 +MOVJ EC00404
SMOVL C00405 +MOVJ EC00405
SMOVL C00406 +MOVJ EC00406
SMOVL C00407 +MOVJ EC00407
SMOVL C00408 +MOVJ EC00408
SMOVL C00409 +MOVJ EC00409
SMOVL C00410 +MOVJ EC00410
SMOVL C00411 +MOVJ EC00411
SMOVL C00412 +MOVJ EC00412
SMOVL C00413 +MOVJ EC00413
SMOVL C00414 +MOVJ EC00414
SMOVL C00415 +MOVJ EC00415
SMOVL C00416 +MOVJ EC00416
SMOVL C00417 +MOVJ EC00417
SMOVL C00418 +MOVJ EC00418
SMOVL C00419 +MOVJ EC00419
SMOVL C00420 +MOVJ EC00420
SMOVL C00421 +MOVJ EC00421
SMOVL C00422 +MOVJ EC00422
SMOVL C00423 +MOVJ EC00423
SMOVL C00424 +MOVJ EC00424
SMOVL C00425 +MOVJ EC00425
SMOVL C00426 +MOVJ EC00426
SMOVL C00427 +MOVJ EC00427
SMOVL C00428 +MOVJ EC00428
SMOVL C00429 +MOVJ EC00429
SMOVL C00430 +MOVJ EC00430
SMOVL C00431 +MOVJ EC00431
SMOVL C00432 +MOVJ EC00432
SMOVL C00433 +MOVJ EC00433
SMOVL C00434 +MOVJ EC00434
SMOVL C00435 +MOVJ EC00435
SMOVL C00436 +MOVJ EC00436
SMOVL C00437 +MOVJ EC00437
SMOVL C00438 +MOVJ EC00438
SMOVL C00439 +MOVJ EC00439
SMOVL C00440 +MOVJ EC00440
SMOVL C00441 +MOVJ EC00441
SMOVL C00442 +MOVJ EC00442
SMOVL C00443 +MOVJ EC00443
SMOVL C00444 +MOVJ EC00444
SMOVL C00445 +MOVJ EC00445
SMOVL C00446 +MOVJ EC00446
SMOVL C00447 +MOVJ EC00447
SMOVL C00448 +MOVJ EC00448
SMOVL C00449 +MOVJ EC00449
SMOVL C00450 +MOVJ EC00450
SMOVL C00451 +MOVJ EC00451
SMOVL C00452 +MOVJ EC00452
SMOVL C00453 +MOVJ EC00453
SMOVL C00454 +MOVJ EC00454
SMOVL C00455 +MOVJ EC00455
SMOVL C00456 +MOVJ EC00456
SMOVL C00457 +MOVJ EC00457
SMOVL C00458 +MOVJ EC00458
SMOVL C00459 +MOVJ EC00459
SMOVL C00460 +MOVJ EC00460
SMOVL C00461 +MOVJ EC00461
SMOVL C00462 +MOVJ EC00462
SMOVL C00463 +MOVJ EC00463
SMOVL C00464 +MOVJ EC00464
SMOVL C00465 +MOVJ EC00465
SMOVL C00466 +MOVJ EC00466
SMOVL C00467 +MOVJ EC00467
SMOVL C00468 +MOVJ EC00468
SMOVL C00469 +MOVJ EC00469
SMOVL C00470 +MOVJ EC00470
SMOVL C00471 +MOVJ EC00471
SMOVL C00472 +MOVJ EC00472
SMOVL C00473 +MOVJ EC00473
SMOVL C00474 +MOVJ EC00474
SMOVL C00475 +MOVJ EC00475
SMOVL C00476 +MOVJ EC00476
SMOVL C00477 +MOVJ EC00477
SMOVL C00478 +MOVJ EC00478
SMOVL C00479 +MOVJ EC00479
SMOVL C00480 +MOVJ EC00480
SMOVL C00481 +MOVJ EC00481
SMOVL C00482 +MOVJ EC00482
SMOVL C00483 +MOVJ EC00483
SMOVL C00484 +MOVJ EC00484
SMOVL C00485 +MOVJ EC00485
SMOVL C00486 +MOVJ EC00486
SMOVL C00487 +MOVJ EC00487
SMOVL C00488 +MOVJ EC00488
SMOVL C00489 +MOVJ EC00489
SMOVL C00490 +MOVJ EC00490
SMOVL C00491 +MOVJ EC00491
SMOVL C00492 +MOVJ EC00492
SMOVL C00493 +MOVJ EC00493
SMOVL C00494 +MOVJ EC00494
SMOVL C00495 +MOVJ EC00495
SMOVL C00496 +MOVJ EC00496
SMOVL C00497 +MOVJ EC00497
SMOVL C00498 +MOVJ EC00498
SMOVL C00499 +MOVJ EC00499
SMOVL C00500 +MOVJ EC00500
SMOVL C00501 +MOVJ EC00501
SMOVL C00502 +MOVJ EC00502
SMOVL C00503 +MOVJ EC00503
SMOVL C00504 +MOVJ EC00504
SMOVL C00505 +MOVJ EC00505
SMOVL C00506 +MOVJ EC00506
SMOVL C00507 +MOVJ EC00507
SMOVL C00508 +MOVJ EC00508
SMOVL C00509 +MOVJ EC00509
SMOVL C00510 +MOVJ EC00510
SMOVL C00511 +MOVJ EC00511
SMOVL C00512 +MOVJ EC00512
SMOVL C00513 +MOVJ EC00513
SMOVL C00514 +MOVJ EC00514
SMOVL C00515 +MOVJ EC00515
SMOVL C00516 +MOVJ EC00516
SMOVL C00517 +MOVJ EC00517
SMOVL C00518 +MOVJ EC00518
SMOVL C00519 +MOVJ EC00519
SMOVL C00520 +MOVJ EC00520
SMOVL C00521 +MOVJ EC00521
SMOVL C00522 +MOVJ EC00522
SMOVL C00523 +MOVJ EC00523
SMOVL C00524 +MOVJ EC00524
SMOVL C00525 +MOVJ EC00525
SMOVL C00526 +MOVJ EC00526
SMOVL C00527 +MOVJ EC00527
SMOVL C00528 +MOVJ EC00528
SMOVL C00529 +MOVJ EC00529
SMOVL C00530 +MOVJ EC00530
SMOVL C00531 +MOVJ EC00531
SMOVL C00532 +MOVJ EC00532
SMOVL C00533 +MOVJ EC00533
SMOVL C00534 +MOVJ EC00534
SMOVL C00535 +MOVJ EC00535
SMOVL C00536 +MOVJ EC00536
SMOVL C00537 +MOVJ EC00537
SMOVL C00538 +MOVJ EC00538
SMOVL C00539 +MOVJ EC00539
SMOVL C00540 +MOVJ EC00540
SMOVL C00541 +MOVJ EC00541
SMOVL C00542 +MOVJ EC00542
SMOVL C00543 +MOVJ EC00543
SMOVL C00544 +MOVJ EC00544
SMOVL C00545 +MOVJ EC00545
SMOVL C00546 +MOVJ EC00546
SMOVL C00547 +MOVJ EC00547
SMOVL C00548 +MOVJ EC00548
SMOVL C00549 +MOVJ EC00549
SMOVL C00550 +MOVJ EC00550
SMOVL C00551 +MOVJ EC00551
SMOVL C00552 +MOVJ EC00552
SMOVL C00553 +MOVJ EC00553
SMOVL C00554 +MOVJ EC00554
SMOVL C00555 +MOVJ EC00555
SMOVL C00556 +MOVJ EC00556
SMOVL C00557 +MOVJ EC00557
SMOVL C00558 +MOVJ EC00558
SMOVL C00559 +MOVJ EC00559
SMOVL C00560 +MOVJ EC00560
SMOVL C00561 +MOVJ EC00561
SMOVL C00562 +MOVJ EC00562
SMOVL C00563 +MOVJ EC00563
SMOVL C00564 +MOVJ EC00564
SMOVL C00565 +MOVJ EC00565
SMOVL C00566 +MOVJ EC00566
SMOVL C00567 +MOVJ EC00567
SMOVL C00568 +MOVJ EC00568
SMOVL C00569 +MOVJ EC00569
SMOVL C00570 +MOVJ EC00570
SMOVL C00571 +MOVJ EC00571
SMOVL C00572 +MOVJ EC00572
SMOVL C00573 +MOVJ EC00573
SMOVL C00574 +MOVJ EC00574
SMOVL C00575 +MOVJ EC00575
SMOVL C00576 +MOVJ EC00576
SMOVL C00577 +MOVJ EC00577
SMOVL C00578 +MOVJ EC00578
SMOVL C00579 +MOVJ EC00579
SMOVL C00580 +MOVJ EC00580
SMOVL C00581 +MOVJ EC00581
SMOVL C00582 +MOVJ EC00582
SMOVL C00583 +MOVJ EC00583
SMOVL C00584 +MOVJ EC00584
SMOVL C00585 +MOVJ EC00585
SMOVL C00586 +MOVJ EC00586
SMOVL C00587 +MOVJ EC00587
SMOVL C00588 +MOVJ EC00588
SMOVL C00589 +MOVJ EC00589
SMOVL C00590 +MOVJ EC00590
SMOVL C00591 +MOVJ EC00591
SMOVL C00592 +MOVJ EC00592
SMOVL C00593 +MOVJ EC00593
SMOVL C00594 +MOVJ EC00594
SMOVL C00595 +MOVJ EC00595
SMOVL C00596 +MOVJ EC00596
SMOVL C00597 +MOVJ EC00597
SMOVL C00598 +MOVJ EC00598
SMOVL C00599 +MOVJ EC00599
SMOVL C00600 +MOVJ EC00600
SMOVL C00601 +MOVJ EC00601
SMOVL C00602 +MOVJ EC00602
SMOVL C00603 +MOVJ EC00603
SMOVL C00604 +MOVJ EC00604
SMOVL C00605 +MOVJ EC00605
SMOVL C00606 +MOVJ EC00606
SMOVL C00607 +MOVJ EC00607
SMOVL C00608 +MOVJ EC00608
SMOVL C00609 +MOVJ EC00609
SMOVL C00610 +MOVJ EC00610
SMOVL C00611 +MOVJ EC00611
SMOVL C00612 +MOVJ EC00612
SMOVL C00613 +MOVJ EC00613
SMOVL C00614 +MOVJ EC00614
SMOVL C00615 +MOVJ EC00615
SMOVL C00616 +MOVJ EC00616
SMOVL C00617 +MOVJ EC00617
SMOVL C00618 +MOVJ EC00618
SMOVL C00619 +MOVJ EC00619
SMOVL C00620 +MOVJ EC00620
SMOVL C00621 +MOVJ EC00621
SMOVL C00622 +MOVJ EC00622
SMOVL C00623 +MOVJ EC00623
SMOVL C00624 +MOVJ EC00624
SMOVL C00625 +MOVJ EC00625
SMOVL C00626 +MOVJ EC00626
SMOVL C00627 +MOVJ EC00627
SMOVL C00628 +MOVJ EC00628
SMOVL C00629 +MOVJ EC00629
SMOVL C00630 +MOVJ EC00630
SMOVL C00631 +MOVJ EC00631
SMOVL C00632 +MOVJ EC00632
SMOVL C00633 +MOVJ EC00633
SMOVL C00634 +MOVJ EC00634
SMOVL C00635 +MOVJ EC00635
SMOVL C00636 +MOVJ EC00636
SMOVL C00637 +MOVJ EC00637
SMOVL C00638 +MOVJ EC00638
SMOVL C00639 +MOVJ EC00639
SMOVL C00640 +MOVJ EC00640
SMOVL C00641 +MOVJ EC00641
SMOVL C00642 +MOVJ EC00642
SMOVL C00643 +MOVJ EC00643
SMOVL C00644 +MOVJ EC00644
SMOVL C00645 +MOVJ EC00645
SMOVL C00646 +MOVJ EC00646
SMOVL C00647 +MOVJ EC00647
SMOVL C00648 +MOVJ EC00648
SMOVL C00649 +MOVJ EC00649
SMOVL C00650 +MOVJ EC00650
SMOVL C00651 +MOVJ EC00651
SMOVL C00652 +MOVJ EC00652
SMOVL C00653 +MOVJ EC00653
SMOVL C00654 +MOVJ EC00654
SMOVL C00655 +MOVJ EC00655
SMOVL C00656 +MOVJ EC00656
SMOVL C00657 +MOVJ EC00657
SMOVL C00658 +MOVJ EC00658
SMOVL C00659 +MOVJ EC00659
SMOVL C00660 +MOVJ EC00660
SMOVL C00661 +MOVJ EC00661
SMOVL C00662 +MOVJ EC00662
SMOVL C00663 +MOVJ EC00663
SMOVL C00664 +MOVJ EC00664
SMOVL C00665 +MOVJ EC00665
SMOVL C00666 +MOVJ EC00666
SMOVL C00667 +MOVJ EC00667
SMOVL C00668 +MOVJ EC00668
SMOVL C00669 +MOVJ EC00669
SMOVL C00670 +MOVJ EC00670
SMOVL C00671 +MOVJ EC00671
SMOVL C00672 +MOVJ EC00672
SMOVL C00673 +MOVJ EC00673
SMOVL C00674 +MOVJ EC00674
SMOVL C00675 +MOVJ EC00675
SMOVL C00676 +MOVJ EC00676
SMOVL C00677 +MOVJ EC00677
SMOVL C00678 +MOVJ EC00678
SMOVL C00679 +MOVJ EC00679
SMOVL C00680 +MOVJ EC00680
SMOVL C00681 +MOVJ EC00681
SMOVL C00682 +MOVJ EC00682
SMOVL C00683 +MOVJ EC00683
SMOVL C00684 +MOVJ EC00684
SMOVL C00685 +MOVJ EC00685
SMOVL C00686 +MOVJ EC00686
SMOVL C00687 +MOVJ EC00687
SMOVL C00688 +MOVJ EC00688
SMOVL C00689 +MOVJ EC00689
SMOVL C00690 +MOVJ EC00690
SMOVL C00691 +MOVJ EC00691
SMOVL C00692 +MOVJ EC00692
SMOVL C00693 +MOVJ EC00693
SMOVL C00694 +MOVJ EC00694
SMOVL C00695 +MOVJ EC00695
SMOVL C00696 +MOVJ EC00696
SMOVL C00697 +MOVJ EC00697
SMOVL C00698 +MOVJ EC00698
SMOVL C00699 +MOVJ EC00699
SMOVL C00700 +MOVJ EC00700
SMOVL C00701 +MOVJ EC00701
SMOVL C00702 +MOVJ EC00702
SMOVL C00703 +MOVJ EC00703
SMOVL C00704 +MOVJ EC00704
SMOVL C00705 +MOVJ EC00705
SMOVL C00706 +MOVJ EC00706
SMOVL C00707 +MOVJ EC00707
SMOVL C00708 +MOVJ EC00708
SMOVL C00709 +MOVJ EC00709
SMOVL C00710 +MOVJ EC00710
SMOVL C00711 +MOVJ EC00711
SMOVL C00712 +MOVJ EC00712
SMOVL C00713 +MOVJ EC00713
SMOVL C00714 +MOVJ EC00714
SMOVL C00715 +MOVJ EC00715
SMOVL C00716 +MOVJ EC00716
SMOVL C00717 +MOVJ EC00717
SMOVL C00718 +MOVJ EC00718
SMOVL C00719 +MOVJ EC00719
SMOVL C00720 +MOVJ EC00720
SMOVL C00721 +MOVJ EC00721
SMOVL C00722 +MOVJ EC00722
SMOVL C00723 +MOVJ EC00723
SMOVL C00724 +MOVJ EC00724
SMOVL C00725 +MOVJ EC00725
SMOVL C00726 +MOVJ EC00726
SMOVL C00727 +MOVJ EC00727
SMOVL C00728 +MOVJ EC00728
SMOVL C00729 +MOVJ EC00729
SMOVL C00730 +MOVJ EC00730
SMOVL C00731 +MOVJ EC00731
SMOVL C00732 +MOVJ EC00732
SMOVL C00733 +MOVJ EC00733
SMOVL C00734 +MOVJ EC00734
SMOVL C00735 +MOVJ EC00735
SMOVL C00736 +MOVJ EC00736
SMOVL C00737 +MOVJ EC00737
SMOVL C00738 +MOVJ EC00738
SMOVL C00739 +MOVJ EC00739
SMOVL C00740 +MOVJ EC00740
SMOVL C00741 +MOVJ EC00741
SMOVL C00742 +MOVJ EC00742
SMOVL C00743 +MOVJ EC00743
SMOVL C00744 +MOVJ EC00744
SMOVL C00745 +MOVJ EC00745
SMOVL C00746 +MOVJ EC00746
SMOVL C00747 +MOVJ EC00747
SMOVL C00748 +MOVJ EC00748
SMOVL C00749 +MOVJ EC00749
SMOVL C00750 +MOVJ EC00750
SMOVL C00751 +MOVJ EC00751
SMOVL C00752 +MOVJ EC00752
SMOVL C00753 +MOVJ EC00753
SMOVL C00754 +MOVJ EC00754
SMOVL C00755 +MOVJ EC00755
SMOVL C00756 +MOVJ EC00756
SMOVL C00757 +MOVJ EC00757
SMOVL C00758 +MOVJ EC00758
SMOVL C00759 +MOVJ EC00759
SMOVL C00760 +MOVJ EC00760
SMOVL C00761 +MOVJ EC00761
SMOVL C00762 +MOVJ EC00762
SMOVL C00763 +MOVJ EC00763
SMOVL C00764 +MOVJ EC00764
SMOVL C00765 +MOVJ EC00765
SMOVL C00766 +MOVJ EC00766
SMOVL C00767 +MOVJ EC00767
SMOVL C00768 +MOVJ EC00768
SMOVL C00769 +MOVJ EC00769
SMOVL C00770 +MOVJ EC00770
SMOVL C00771 +MOVJ EC00771
SMOVL C00772 +MOVJ EC00772
SMOVL C00773 +MOVJ EC00773
SMOVL C00774 +MOVJ EC00774
SMOVL C00775 +MOVJ EC00775
SMOVL C00776 +MOVJ EC00776
SMOVL C00777 +MOVJ EC00777
SMOVL C00778 +MOVJ EC00778
SMOVL C00779 +MOVJ EC00779
SMOVL C00780 +MOVJ EC00780
SMOVL C00781 +MOVJ EC00781
SMOVL C00782 +MOVJ EC00782
SMOVL C00783 +MOVJ EC00783
SMOVL C00784 +MOVJ EC00784
SMOVL C00785 +MOVJ EC00785
SMOVL C00786 +MOVJ EC00786
SMOVL C00787 +MOVJ EC00787
SMOVL C00788 +MOVJ EC00788
SMOVL C00789 +MOVJ EC00789
SMOVL C00790 +MOVJ EC00790
SMOVL C00791 +MOVJ EC00791
SMOVL C00792 +MOVJ EC00792
SMOVL C00793 +MOVJ EC00793
SMOVL C00794 +MOVJ EC00794
SMOVL C00795 +MOVJ EC00795
SMOVL C00796 +MOVJ EC00796
SMOVL C00797 +MOVJ EC00797
SMOVL C00798 +MOVJ EC00798
SMOVL C00799 +MOVJ EC00799
SMOVL C00800 +MOVJ EC00800
SMOVL C00801 +MOVJ EC00801
SMOVL C00802 +MOVJ EC00802
SMOVL C00803 +MOVJ EC00803
SMOVL C00804 +MOVJ EC00804
SMOVL C00805 +MOVJ EC00805
SMOVL C00806 +MOVJ EC00806
SMOVL C00807 +MOVJ EC00807
SMOVL C00808 +MOVJ EC00808
SMOVL C00809 +MOVJ EC00809
SMOVL C00810 +MOVJ EC00810
SMOVL C00811 +MOVJ EC00811
SMOVL C00812 +MOVJ EC00812
SMOVL C00813 +MOVJ EC00813
SMOVL C00814 +MOVJ EC00814
SMOVL C00815 +MOVJ EC00815
SMOVL C00816 +MOVJ EC00816
SMOVL C00817 +MOVJ EC00817
SMOVL C00818 +MOVJ EC00818
SMOVL C00819 +MOVJ EC00819
SMOVL C00820 +MOVJ EC00820
SMOVL C00821 +MOVJ EC00821
SMOVL C00822 +MOVJ EC00822
SMOVL C00823 +MOVJ EC00823
SMOVL C00824 +MOVJ EC00824
SMOVL C00825 +MOVJ EC00825
SMOVL C00826 +MOVJ EC00826
SMOVL C00827 +MOVJ EC00827
SMOVL C00828 +MOVJ EC00828
SMOVL C00829 +MOVJ EC00829
SMOVL C00830 +MOVJ EC00830
SMOVL C00831 +MOVJ EC00831
SMOVL C00832 +MOVJ EC00832
SMOVL C00833 +MOVJ EC00833
SMOVL C00834 +MOVJ EC00834
SMOVL C00835 +MOVJ EC00835
SMOVL C00836 +MOVJ EC00836
SMOVL C00837 +MOVJ EC00837
SMOVL C00838 +MOVJ EC00838
SMOVL C00839 +MOVJ EC00839
SMOVL C00840 +MOVJ EC00840
SMOVL C00841 +MOVJ EC00841
SMOVL C00842 +MOVJ EC00842
SMOVL C00843 +MOVJ EC00843
SMOVL C00844 +MOVJ EC00844
SMOVL C00845 +MOVJ EC00845
SMOVL C00846 +MOVJ EC00846
SMOVL C00847 +MOVJ EC00847
SMOVL C00848 +MOVJ EC00848
SMOVL C00849 +MOVJ EC00849
SMOVL C00850 +MOVJ EC00850
SMOVL C00851 +MOVJ EC00851
SMOVL C00852 +MOVJ EC00852
SMOVL C00853 +MOVJ EC00853
SMOVL C00854 +MOVJ EC00854
SMOVL C00855 +MOVJ EC00855
SMOVL C00856 +MOVJ EC00856
SMOVL C00857 +MOVJ EC00857
SMOVL C00858 +MOVJ EC00858
SMOVL C00859 +MOVJ EC00859
SMOVL C00860 +MOVJ EC00860
SMOVL C00861 +MOVJ EC00861
SMOVL C00862 +MOVJ EC00862
SMOVL C00863 +MOVJ EC00863
SMOVL C00864 +MOVJ EC00864
SMOVL C00865 +MOVJ EC00865
SMOVL C00866 +MOVJ EC00866
SMOVL C00867 +MOVJ EC00867
SMOVL C00868 +MOVJ EC00868
SMOVL C00869 +MOVJ EC00869
SMOVL C00870 +MOVJ EC00870
SMOVL C00871 +MOVJ EC00871
SMOVL C00872 +MOVJ EC00872
SMOVL C00873 +MOVJ EC00873
SMOVL C00874 +MOVJ EC00874
SMOVL C00875 +MOVJ EC00875
SMOVL C00876 +MOVJ EC00876
SMOVL C00877 +MOVJ EC00877
SMOVL C00878 +MOVJ EC00878
SMOVL C00879 +MOVJ EC00879
SMOVL C00880 +MOVJ EC00880
SMOVL C00881 +MOVJ EC00881
SMOVL C00882 +MOVJ EC00882
SMOVL C00883 +MOVJ EC00883
SMOVL C00884 +MOVJ EC00884
SMOVL C00885 +MOVJ EC00885
SMOVL C00886 +MOVJ EC00886
SMOVL C00887 +MOVJ EC00887
SMOVL C00888 +MOVJ EC00888
SMOVL C00889 +MOVJ EC00889
SMOVL C00890 +MOVJ EC00890
SMOVL C00891 +MOVJ EC00891
SMOVL C00892 +MOVJ EC00892
SMOVL C00893 +MOVJ EC00893
SMOVL C00894 +MOVJ EC00894
SMOVL C00895 +MOVJ EC00895
SMOVL C00896 +MOVJ EC00896
SMOVL C00897 +MOVJ EC00897
ARCOF
SMOVL C00898 +MOVJ EC00898
ARCON
SMOVL C00899 +MOVJ EC00899
SMOVL C00900 +MOVJ EC00900
SMOVL C00901 +MOVJ EC00901
SMOVL C00902 +MOVJ EC00902
SMOVL C00903 +MOVJ EC00903
SMOVL C00904 +MOVJ EC00904
SMOVL C00905 +MOVJ EC00905
SMOVL C00906 +MOVJ EC00906
SMOVL C00907 +MOVJ EC00907
SMOVL C00908 +MOVJ EC00908
SMOVL C00909 +MOVJ EC00909
SMOVL C00910 +MOVJ EC00910
SMOVL C00911 +MOVJ EC00911
SMOVL C00912 +MOVJ EC00912
SMOVL C00913 +MOVJ EC00913
SMOVL C00914 +MOVJ EC00914
SMOVL C00915 +MOVJ EC00915
SMOVL C00916 +MOVJ EC00916
ARCOF
SMOVL C00917 +MOVJ EC00917
ARCON
SMOVL C00918 +MOVJ EC00918
SMOVL C00919 +MOVJ EC00919
SMOVL C00920 +MOVJ EC00920
SMOVL C00921 +MOVJ EC00921
SMOVL C00922 +MOVJ EC00922
SMOVL C00923 +MOVJ EC00923
SMOVL C00924 +MOVJ EC00924
SMOVL C00925 +MOVJ EC00925
SMOVL C00926 +MOVJ EC00926
SMOVL C00927 +MOVJ EC00927
SMOVL C00928 +MOVJ EC00928
SMOVL C00929 +MOVJ EC00929
SMOVL C00930 +MOVJ EC00930
SMOVL C00931 +MOVJ EC00931
SMOVL C00932 +MOVJ EC00932
SMOVL C00933 +MOVJ EC00933
SMOVL C00934 +MOVJ EC00934
SMOVL C00935 +MOVJ EC00935
ARCOF
SMOVL C00936 +MOVJ EC00936
ARCON
SMOVL C00937 +MOVJ EC00937
SMOVL C00938 +MOVJ EC00938
SMOVL C00939 +MOVJ EC00939
SMOVL C00940 +MOVJ EC00940
SMOVL C00941 +MOVJ EC00941
SMOVL C00942 +MOVJ EC00942
SMOVL C00943 +MOVJ EC00943
SMOVL C00944 +MOVJ EC00944
SMOVL C00945 +MOVJ EC00945
SMOVL C00946 +MOVJ EC00946
SMOVL C00947 +MOVJ EC00947
SMOVL C00948 +MOVJ EC00948
SMOVL C00949 +MOVJ EC00949
SMOVL C00950 +MOVJ EC00950
SMOVL C00951 +MOVJ EC00951
SMOVL C00952 +MOVJ EC00952
SMOVL C00953 +MOVJ EC00953
SMOVL C00954 +MOVJ EC00954
ARCOF
SMOVL C00955 +MOVJ EC00955
ARCON
SMOVL C00956 +MOVJ EC00956
SMOVL C00957 +MOVJ EC00957
SMOVL C00958 +MOVJ EC00958
SMOVL C00959 +MOVJ EC00959
SMOVL C00960 +MOVJ EC00960
SMOVL C00961 +MOVJ EC00961
SMOVL C00962 +MOVJ EC00962
SMOVL C00963 +MOVJ EC00963
SMOVL C00964 +MOVJ EC00964
SMOVL C00965 +MOVJ EC00965
SMOVL C00966 +MOVJ EC00966
SMOVL C00967 +MOVJ EC00967
SMOVL C00968 +MOVJ EC00968
SMOVL C00969 +MOVJ EC00969
SMOVL C00970 +MOVJ EC00970
SMOVL C00971 +MOVJ EC00971
SMOVL C00972 +MOVJ EC00972
SMOVL C00973 +MOVJ EC00973
SMOVL C00974 +MOVJ EC00974
ARCOF
SMOVL C00975 +MOVJ EC00975
ARCON
SMOVL C00976 +MOVJ EC00976
SMOVL C00977 +MOVJ EC00977
SMOVL C00978 +MOVJ EC00978
SMOVL C00979 +MOVJ EC00979
SMOVL C00980 +MOVJ EC00980
SMOVL C00981 +MOVJ EC00981
SMOVL C00982 +MOVJ EC00982
SMOVL C00983 +MOVJ EC00983
SMOVL C00984 +MOVJ EC00984
SMOVL C00985 +MOVJ EC00985
SMOVL C00986 +MOVJ EC00986
SMOVL C00987 +MOVJ EC00987
SMOVL C00988 +MOVJ EC00988
SMOVL C00989 +MOVJ EC00989
SMOVL C00990 +MOVJ EC00990
SMOVL C00991 +MOVJ EC00991
SMOVL C00992 +MOVJ EC00992
SMOVL C00993 +MOVJ EC00993
ARCOF
SMOVL C00994 +MOVJ EC00994
ARCON
SMOVL C00995 +MOVJ EC00995
SMOVL C00996 +MOVJ EC00996
SMOVL C00997 +MOVJ EC00997
SMOVL C00998 +MOVJ EC00998
SMOVL C00999 +MOVJ EC00999
SMOVL C01000 +MOVJ EC01000
SMOVL C01001 +MOVJ EC01001
SMOVL C01002 +MOVJ EC01002
SMOVL C01003 +MOVJ EC01003
SMOVL C01004 +MOVJ EC01004
SMOVL C01005 +MOVJ EC01005
SMOVL C01006 +MOVJ EC01006
SMOVL C01007 +MOVJ EC01007
SMOVL C01008 +MOVJ EC01008
SMOVL C01009 +MOVJ EC01009
SMOVL C01010 +MOVJ EC01010
SMOVL C01011 +MOVJ EC01011
SMOVL C01012 +MOVJ EC01012
ARCOF
SMOVL C01013 +MOVJ EC01013
ARCON
SMOVL C01014 +MOVJ EC01014
SMOVL C01015 +MOVJ EC01015
SMOVL C01016 +MOVJ EC01016
SMOVL C01017 +MOVJ EC01017
SMOVL C01018 +MOVJ EC01018
SMOVL C01019 +MOVJ EC01019
SMOVL C01020 +MOVJ EC01020
SMOVL C01021 +MOVJ EC01021
SMOVL C01022 +MOVJ EC01022
SMOVL C01023 +MOVJ EC01023
SMOVL C01024 +MOVJ EC01024
SMOVL C01025 +MOVJ EC01025
SMOVL C01026 +MOVJ EC01026
SMOVL C01027 +MOVJ EC01027
SMOVL C01028 +MOVJ EC01028
SMOVL C01029 +MOVJ EC01029
SMOVL C01030 +MOVJ EC01030
SMOVL C01031 +MOVJ EC01031
ARCOF
SMOVL C01032 +MOVJ EC01032
ARCON
SMOVL C01033 +MOVJ EC01033
SMOVL C01034 +MOVJ EC01034
SMOVL C01035 +MOVJ EC01035
SMOVL C01036 +MOVJ EC01036
SMOVL C01037 +MOVJ EC01037
SMOVL C01038 +MOVJ EC01038
SMOVL C01039 +MOVJ EC01039
SMOVL C01040 +MOVJ EC01040
SMOVL C01041 +MOVJ EC01041
SMOVL C01042 +MOVJ EC01042
SMOVL C01043 +MOVJ EC01043
SMOVL C01044 +MOVJ EC01044
SMOVL C01045 +MOVJ EC01045
SMOVL C01046 +MOVJ EC01046
SMOVL C01047 +MOVJ EC01047
SMOVL C01048 +MOVJ EC01048
ARCOF
SMOVL C01049 +MOVJ EC01049
ARCON
SMOVL C01050 +MOVJ EC01050
SMOVL C01051 +MOVJ EC01051
SMOVL C01052 +MOVJ EC01052
SMOVL C01053 +MOVJ EC01053
SMOVL C01054 +MOVJ EC01054
SMOVL C01055 +MOVJ EC01055
SMOVL C01056 +MOVJ EC01056
SMOVL C01057 +MOVJ EC01057
SMOVL C01058 +MOVJ EC01058
SMOVL C01059 +MOVJ EC01059
SMOVL C01060 +MOVJ EC01060
SMOVL C01061 +MOVJ EC01061
ARCOF
SMOVL C01062 +MOVJ EC01062
ARCON
SMOVL C01063 +MOVJ EC01063
SMOVL C01064 +MOVJ EC01064
SMOVL C01065 +MOVJ EC01065
SMOVL C01066 +MOVJ EC01066
SMOVL C01067 +MOVJ EC01067
SMOVL C01068 +MOVJ EC01068
SMOVL C01069 +MOVJ EC01069
SMOVL C01070 +MOVJ EC01070
SMOVL C01071 +MOVJ EC01071
SMOVL C01072 +MOVJ EC01072
SMOVL C01073 +MOVJ EC01073
SMOVL C01074 +MOVJ EC01074
ARCOF
SMOVL C01075 +MOVJ EC01075
ARCON
SMOVL C01076 +MOVJ EC01076
SMOVL C01077 +MOVJ EC01077
SMOVL C01078 +MOVJ EC01078
SMOVL C01079 +MOVJ EC01079
SMOVL C01080 +MOVJ EC01080
SMOVL C01081 +MOVJ EC01081
SMOVL C01082 +MOVJ EC01082
SMOVL C01083 +MOVJ EC01083
SMOVL C01084 +MOVJ EC01084
SMOVL C01085 +MOVJ EC01085
SMOVL C01086 +MOVJ EC01086
SMOVL C01087 +MOVJ EC01087
ARCOF
SMOVL C01088 +MOVJ EC01088
ARCON
SMOVL C01089 +MOVJ EC01089
SMOVL C01090 +MOVJ EC01090
SMOVL C01091 +MOVJ EC01091
SMOVL C01092 +MOVJ EC01092
SMOVL C01093 +MOVJ EC01093
SMOVL C01094 +MOVJ EC01094
SMOVL C01095 +MOVJ EC01095
SMOVL C01096 +MOVJ EC01096
SMOVL C01097 +MOVJ EC01097
SMOVL C01098 +MOVJ EC01098
SMOVL C01099 +MOVJ EC01099
SMOVL C01100 +MOVJ EC01100
SMOVL C01101 +MOVJ EC01101
ARCOF
SMOVL C01102 +MOVJ EC01102
ARCON
SMOVL C01103 +MOVJ EC01103
SMOVL C01104 +MOVJ EC01104
SMOVL C01105 +MOVJ EC01105
SMOVL C01106 +MOVJ EC01106
SMOVL C01107 +MOVJ EC01107
SMOVL C01108 +MOVJ EC01108
SMOVL C01109 +MOVJ EC01109
SMOVL C01110 +MOVJ EC01110
SMOVL C01111 +MOVJ EC01111
SMOVL C01112 +MOVJ EC01112
SMOVL C01113 +MOVJ EC01113
SMOVL C01114 +MOVJ EC01114
ARCOF
SMOVL C01115 +MOVJ EC01115
ARCON
SMOVL C01116 +MOVJ EC01116
SMOVL C01117 +MOVJ EC01117
SMOVL C01118 +MOVJ EC01118
SMOVL C01119 +MOVJ EC01119
SMOVL C01120 +MOVJ EC01120
SMOVL C01121 +MOVJ EC01121
SMOVL C01122 +MOVJ EC01122
SMOVL C01123 +MOVJ EC01123
SMOVL C01124 +MOVJ EC01124
SMOVL C01125 +MOVJ EC01125
SMOVL C01126 +MOVJ EC01126
SMOVL C01127 +MOVJ EC01127
ARCOF
SMOVL C01128 +MOVJ EC01128
ARCON
SMOVL C01129 +MOVJ EC01129
SMOVL C01130 +MOVJ EC01130
SMOVL C01131 +MOVJ EC01131
SMOVL C01132 +MOVJ EC01132
SMOVL C01133 +MOVJ EC01133
SMOVL C01134 +MOVJ EC01134
SMOVL C01135 +MOVJ EC01135
SMOVL C01136 +MOVJ EC01136
SMOVL C01137 +MOVJ EC01137
SMOVL C01138 +MOVJ EC01138
SMOVL C01139 +MOVJ EC01139
SMOVL C01140 +MOVJ EC01140
ARCOF
SMOVL C01141 +MOVJ EC01141
ARCON
SMOVL C01142 +MOVJ EC01142
SMOVL C01143 +MOVJ EC01143
SMOVL C01144 +MOVJ EC01144
SMOVL C01145 +MOVJ EC01145
SMOVL C01146 +MOVJ EC01146
SMOVL C01147 +MOVJ EC01147
SMOVL C01148 +MOVJ EC01148
SMOVL C01149 +MOVJ EC01149
SMOVL C01150 +MOVJ EC01150
SMOVL C01151 +MOVJ EC01151
SMOVL C01152 +MOVJ EC01152
SMOVL C01153 +MOVJ EC01153
ARCOF
SMOVL C01154 +MOVJ EC01154
ARCON
SMOVL C01155 +MOVJ EC01155
SMOVL C01156 +MOVJ EC01156
SMOVL C01157 +MOVJ EC01157
SMOVL C01158 +MOVJ EC01158
SMOVL C01159 +MOVJ EC01159
SMOVL C01160 +MOVJ EC01160
SMOVL C01161 +MOVJ EC01161
SMOVL C01162 +MOVJ EC01162
SMOVL C01163 +MOVJ EC01163
SMOVL C01164 +MOVJ EC01164
ARCOF
SMOVL C01165 +MOVJ EC01165
ARCON
SMOVL C01166 +MOVJ EC01166
SMOVL C01167 +MOVJ EC01167
SMOVL C01168 +MOVJ EC01168
SMOVL C01169 +MOVJ EC01169
SMOVL C01170 +MOVJ EC01170
SMOVL C01171 +MOVJ EC01171
SMOVL C01172 +MOVJ EC01172
SMOVL C01173 +MOVJ EC01173
SMOVL C01174 +MOVJ EC01174
SMOVL C01175 +MOVJ EC01175
ARCOF
SMOVL C01176 +MOVJ EC01176
ARCON
SMOVL C01177 +MOVJ EC01177
SMOVL C01178 +MOVJ EC01178
SMOVL C01179 +MOVJ EC01179
SMOVL C01180 +MOVJ EC01180
SMOVL C01181 +MOVJ EC01181
SMOVL C01182 +MOVJ EC01182
SMOVL C01183 +MOVJ EC01183
SMOVL C01184 +MOVJ EC01184
SMOVL C01185 +MOVJ EC01185
SMOVL C01186 +MOVJ EC01186
ARCOF
SMOVL C01187 +MOVJ EC01187
ARCON
SMOVL C01188 +MOVJ EC01188
SMOVL C01189 +MOVJ EC01189
SMOVL C01190 +MOVJ EC01190
SMOVL C01191 +MOVJ EC01191
SMOVL C01192 +MOVJ EC01192
SMOVL C01193 +MOVJ EC01193
SMOVL C01194 +MOVJ EC01194
SMOVL C01195 +MOVJ EC01195
SMOVL C01196 +MOVJ EC01196
SMOVL C01197 +MOVJ EC01197
SMOVL C01198 +MOVJ EC01198
ARCOF
SMOVL C01199 +MOVJ EC01199
ARCON
SMOVL C01200 +MOVJ EC01200
SMOVL C01201 +MOVJ EC01201
SMOVL C01202 +MOVJ EC01202
SMOVL C01203 +MOVJ EC01203
SMOVL C01204 +MOVJ EC01204
SMOVL C01205 +MOVJ EC01205
SMOVL C01206 +MOVJ EC01206
SMOVL C01207 +MOVJ EC01207
SMOVL C01208 +MOVJ EC01208
SMOVL C01209 +MOVJ EC01209
ARCOF
SMOVL C01210 +MOVJ EC01210
ARCON
SMOVL C01211 +MOVJ EC01211
SMOVL C01212 +MOVJ EC01212
SMOVL C01213 +MOVJ EC01213
SMOVL C01214 +MOVJ EC01214
SMOVL C01215 +MOVJ EC01215
SMOVL C01216 +MOVJ EC01216
SMOVL C01217 +MOVJ EC01217
SMOVL C01218 +MOVJ EC01218
SMOVL C01219 +MOVJ EC01219
SMOVL C01220 +MOVJ EC01220
ARCOF
SMOVL C01221 +MOVJ EC01221
ARCON
SMOVL C01222 +MOVJ EC01222
SMOVL C01223 +MOVJ EC01223
SMOVL C01224 +MOVJ EC01224
SMOVL C01225 +MOVJ EC01225
SMOVL C01226 +MOVJ EC01226
SMOVL C01227 +MOVJ EC01227
SMOVL C01228 +MOVJ EC01228
SMOVL C01229 +MOVJ EC01229
SMOVL C01230 +MOVJ EC01230
SMOVL C01231 +MOVJ EC01231
ARCOF
SMOVL C01232 +MOVJ EC01232
ARCON
SMOVL C01233 +MOVJ EC01233
SMOVL C01234 +MOVJ EC01234
SMOVL C01235 +MOVJ EC01235
SMOVL C01236 +MOVJ EC01236
SMOVL C01237 +MOVJ EC01237
SMOVL C01238 +MOVJ EC01238
SMOVL C01239 +MOVJ EC01239
SMOVL C01240 +MOVJ EC01240
SMOVL C01241 +MOVJ EC01241
SMOVL C01242 +MOVJ EC01242
SMOVL C01243 +MOVJ EC01243
ARCOF
SMOVL C01244 +MOVJ EC01244
ARCON
SMOVL C01245 +MOVJ EC01245
SMOVL C01246 +MOVJ EC01246
SMOVL C01247 +MOVJ EC01247
SMOVL C01248 +MOVJ EC01248
SMOVL C01249 +MOVJ EC01249
SMOVL C01250 +MOVJ EC01250
SMOVL C01251 +MOVJ EC01251
SMOVL C01252 +MOVJ EC01252
SMOVL C01253 +MOVJ EC01253
SMOVL C01254 +MOVJ EC01254
ARCOF
SMOVL C01255 +MOVJ EC01255
ARCON
SMOVL C01256 +MOVJ EC01256
SMOVL C01257 +MOVJ EC01257
SMOVL C01258 +MOVJ EC01258
SMOVL C01259 +MOVJ EC01259
SMOVL C01260 +MOVJ EC01260
SMOVL C01261 +MOVJ EC01261
SMOVL C01262 +MOVJ EC01262
SMOVL C01263 +MOVJ EC01263
SMOVL C01264 +MOVJ EC01264
SMOVL C01265 +MOVJ EC01265
ARCOF
SMOVL C01266 +MOVJ EC01266
ARCON
SMOVL C01267 +MOVJ EC01267
SMOVL C01268 +MOVJ EC01268
SMOVL C01269 +MOVJ EC01269
SMOVL C01270 +MOVJ EC01270
SMOVL C01271 +MOVJ EC01271
SMOVL C01272 +MOVJ EC01272
SMOVL C01273 +MOVJ EC01273
SMOVL C01274 +MOVJ EC01274
SMOVL C01275 +MOVJ EC01275
SMOVL C01276 +MOVJ EC01276
ARCOF
SMOVL C01277 +MOVJ EC01277
ARCON
SMOVL C01278 +MOVJ EC01278
SMOVL C01279 +MOVJ EC01279
SMOVL C01280 +MOVJ EC01280
SMOVL C01281 +MOVJ EC01281
SMOVL C01282 +MOVJ EC01282
SMOVL C01283 +MOVJ EC01283
SMOVL C01284 +MOVJ EC01284
SMOVL C01285 +MOVJ EC01285
SMOVL C01286 +MOVJ EC01286
SMOVL C01287 +MOVJ EC01287
SMOVL C01288 +MOVJ EC01288
ARCOF
SMOVL C01289 +MOVJ EC01289
ARCON
SMOVL C01290 +MOVJ EC01290
SMOVL C01291 +MOVJ EC01291
SMOVL C01292 +MOVJ EC01292
SMOVL C01293 +MOVJ EC01293
SMOVL C01294 +MOVJ EC01294
SMOVL C01295 +MOVJ EC01295
SMOVL C01296 +MOVJ EC01296
SMOVL C01297 +MOVJ EC01297
SMOVL C01298 +MOVJ EC01298
SMOVL C01299 +MOVJ EC01299
ARCOF
SMOVL C01300 +MOVJ EC01300
ARCON
SMOVL C01301 +MOVJ EC01301
SMOVL C01302 +MOVJ EC01302
SMOVL C01303 +MOVJ EC01303
SMOVL C01304 +MOVJ EC01304
SMOVL C01305 +MOVJ EC01305
SMOVL C01306 +MOVJ EC01306
SMOVL C01307 +MOVJ EC01307
SMOVL C01308 +MOVJ EC01308
SMOVL C01309 +MOVJ EC01309
SMOVL C01310 +MOVJ EC01310
ARCOF
SMOVL C01311 +MOVJ EC01311
ARCON
SMOVL C01312 +MOVJ EC01312
SMOVL C01313 +MOVJ EC01313
SMOVL C01314 +MOVJ EC01314
SMOVL C01315 +MOVJ EC01315
SMOVL C01316 +MOVJ EC01316
SMOVL C01317 +MOVJ EC01317
SMOVL C01318 +MOVJ EC01318
SMOVL C01319 +MOVJ EC01319
SMOVL C01320 +MOVJ EC01320
SMOVL C01321 +MOVJ EC01321
ARCOF
SMOVL C01322 +MOVJ EC01322
ARCON
SMOVL C01323 +MOVJ EC01323
SMOVL C01324 +MOVJ EC01324
SMOVL C01325 +MOVJ EC01325
SMOVL C01326 +MOVJ EC01326
SMOVL C01327 +MOVJ EC01327
SMOVL C01328 +MOVJ EC01328
SMOVL C01329 +MOVJ EC01329
SMOVL C01330 +MOVJ EC01330
SMOVL C01331 +MOVJ EC01331
SMOVL C01332 +MOVJ EC01332
ARCOF
SMOVL C01333 +MOVJ EC01333
ARCON
SMOVL C01334 +MOVJ EC01334
SMOVL C01335 +MOVJ EC01335
SMOVL C01336 +MOVJ EC01336
SMOVL C01337 +MOVJ EC01337
SMOVL C01338 +MOVJ EC01338
SMOVL C01339 +MOVJ EC01339
SMOVL C01340 +MOVJ EC01340
SMOVL C01341 +MOVJ EC01341
ARCOF
SMOVL C01342 +MOVJ EC01342
ARCON
SMOVL C01343 +MOVJ EC01343
SMOVL C01344 +MOVJ EC01344
SMOVL C01345 +MOVJ EC01345
SMOVL C01346 +MOVJ EC01346
SMOVL C01347 +MOVJ EC01347
SMOVL C01348 +MOVJ EC01348
SMOVL C01349 +MOVJ EC01349
SMOVL C01350 +MOVJ EC01350
ARCOF
SMOVL C01351 +MOVJ EC01351
ARCON
SMOVL C01352 +MOVJ EC01352
SMOVL C01353 +MOVJ EC01353
SMOVL C01354 +MOVJ EC01354
SMOVL C01355 +MOVJ EC01355
SMOVL C01356 +MOVJ EC01356
SMOVL C01357 +MOVJ EC01357
SMOVL C01358 +MOVJ EC01358
SMOVL C01359 +MOVJ EC01359
ARCOF
SMOVL C01360 +MOVJ EC01360
ARCON
SMOVL C01361 +MOVJ EC01361
SMOVL C01362 +MOVJ EC01362
SMOVL C01363 +MOVJ EC01363
SMOVL C01364 +MOVJ EC01364
SMOVL C01365 +MOVJ EC01365
SMOVL C01366 +MOVJ EC01366
SMOVL C01367 +MOVJ EC01367
SMOVL C01368 +MOVJ EC01368
SMOVL C01369 +MOVJ EC01369
ARCOF
SMOVL C01370 +MOVJ EC01370
ARCON
SMOVL C01371 +MOVJ EC01371
SMOVL C01372 +MOVJ EC01372
SMOVL C01373 +MOVJ EC01373
SMOVL C01374 +MOVJ EC01374
SMOVL C01375 +MOVJ EC01375
SMOVL C01376 +MOVJ EC01376
SMOVL C01377 +MOVJ EC01377
SMOVL C01378 +MOVJ EC01378
ARCOF
SMOVL C01379 +MOVJ EC01379
ARCON
SMOVL C01380 +MOVJ EC01380
SMOVL C01381 +MOVJ EC01381
SMOVL C01382 +MOVJ EC01382
SMOVL C01383 +MOVJ EC01383
SMOVL C01384 +MOVJ EC01384
SMOVL C01385 +MOVJ EC01385
SMOVL C01386 +MOVJ EC01386
SMOVL C01387 +MOVJ EC01387
ARCOF
SMOVL C01388 +MOVJ EC01388
ARCON
SMOVL C01389 +MOVJ EC01389
SMOVL C01390 +MOVJ EC01390
SMOVL C01391 +MOVJ EC01391
SMOVL C01392 +MOVJ EC01392
SMOVL C01393 +MOVJ EC01393
SMOVL C01394 +MOVJ EC01394
SMOVL C01395 +MOVJ EC01395
SMOVL C01396 +MOVJ EC01396
ARCOF
SMOVL C01397 +MOVJ EC01397
ARCON
SMOVL C01398 +MOVJ EC01398
SMOVL C01399 +MOVJ EC01399
SMOVL C01400 +MOVJ EC01400
SMOVL C01401 +MOVJ EC01401
SMOVL C01402 +MOVJ EC01402
SMOVL C01403 +MOVJ EC01403
SMOVL C01404 +MOVJ EC01404
SMOVL C01405 +MOVJ EC01405
ARCOF
SMOVL C01406 +MOVJ EC01406
ARCON
SMOVL C01407 +MOVJ EC01407
SMOVL C01408 +MOVJ EC01408
SMOVL C01409 +MOVJ EC01409
SMOVL C01410 +MOVJ EC01410
SMOVL C01411 +MOVJ EC01411
SMOVL C01412 +MOVJ EC01412
ARCOF
SMOVL C01413 +MOVJ EC01413
ARCON
SMOVL C01414 +MOVJ EC01414
SMOVL C01415 +MOVJ EC01415
SMOVL C01416 +MOVJ EC01416
SMOVL C01417 +MOVJ EC01417
SMOVL C01418 +MOVJ EC01418
SMOVL C01419 +MOVJ EC01419
ARCOF
SMOVL C01420 +MOVJ EC01420
ARCON
SMOVL C01421 +MOVJ EC01421
SMOVL C01422 +MOVJ EC01422
SMOVL C01423 +MOVJ EC01423
SMOVL C01424 +MOVJ EC01424
SMOVL C01425 +MOVJ EC01425
SMOVL C01426 +MOVJ EC01426
ARCOF
SMOVL C01427 +MOVJ EC01427
ARCON
SMOVL C01428 +MOVJ EC01428
SMOVL C01429 +MOVJ EC01429
SMOVL C01430 +MOVJ EC01430
SMOVL C01431 +MOVJ EC01431
SMOVL C01432 +MOVJ EC01432
SMOVL C01433 +MOVJ EC01433
SMOVL C01434 +MOVJ EC01434
ARCOF
SMOVL C01435 +MOVJ EC01435
ARCON
SMOVL C01436 +MOVJ EC01436
SMOVL C01437 +MOVJ EC01437
SMOVL C01438 +MOVJ EC01438
SMOVL C01439 +MOVJ EC01439
SMOVL C01440 +MOVJ EC01440
SMOVL C01441 +MOVJ EC01441
ARCOF
SMOVL C01442 +MOVJ EC01442
ARCON
SMOVL C01443 +MOVJ EC01443
SMOVL C01444 +MOVJ EC01444
SMOVL C01445 +MOVJ EC01445
SMOVL C01446 +MOVJ EC01446
SMOVL C01447 +MOVJ EC01447
SMOVL C01448 +MOVJ EC01448
ARCOF
SMOVL C01449 +MOVJ EC01449
ARCON
SMOVL C01450 +MOVJ EC01450
SMOVL C01451 +MOVJ EC01451
SMOVL C01452 +MOVJ EC01452
SMOVL C01453 +MOVJ EC01453
SMOVL C01454 +MOVJ EC01454
SMOVL C01455 +MOVJ EC01455
ARCOF
SMOVL C01456 +MOVJ EC01456
ARCON
SMOVL C01457 +MOVJ EC01457
SMOVL C01458 +MOVJ EC01458
SMOVL C01459 +MOVJ EC01459
SMOVL C01460 +MOVJ EC01460
SMOVL C01461 +MOVJ EC01461
SMOVL C01462 +MOVJ EC01462
SMOVL C01463 +MOVJ EC01463
ARCOF
SMOVL C01464 +MOVJ EC01464
ARCON
SMOVL C01465 +MOVJ EC01465
SMOVL C01466 +MOVJ EC01466
SMOVL C01467 +MOVJ EC01467
SMOVL C01468 +MOVJ EC01468
SMOVL C01469 +MOVJ EC01469
SMOVL C01470 +MOVJ EC01470
ARCOF
SMOVL C01471 +MOVJ EC01471
ARCON
SMOVL C01472 +MOVJ EC01472
SMOVL C01473 +MOVJ EC01473
SMOVL C01474 +MOVJ EC01474
SMOVL C01475 +MOVJ EC01475
SMOVL C01476 +MOVJ EC01476
SMOVL C01477 +MOVJ EC01477
ARCOF
SMOVL C01478 +MOVJ EC01478
ARCON
SMOVL C01479 +MOVJ EC01479
SMOVL C01480 +MOVJ EC01480
SMOVL C01481 +MOVJ EC01481
SMOVL C01482 +MOVJ EC01482
SMOVL C01483 +MOVJ EC01483
SMOVL C01484 +MOVJ EC01484
ARCOF
SMOVL C01485 +MOVJ EC01485
ARCON
SMOVL C01486 +MOVJ EC01486
SMOVL C01487 +MOVJ EC01487
SMOVL C01488 +MOVJ EC01488
SMOVL C01489 +MOVJ EC01489
SMOVL C01490 +MOVJ EC01490
SMOVL C01491 +MOVJ EC01491
SMOVL C01492 +MOVJ EC01492
ARCOF
SMOVL C01493 +MOVJ EC01493
ARCON
SMOVL C01494 +MOVJ EC01494
SMOVL C01495 +MOVJ EC01495
SMOVL C01496 +MOVJ EC01496
SMOVL C01497 +MOVJ EC01497
SMOVL C01498 +MOVJ EC01498
SMOVL C01499 +MOVJ EC01499
ARCOF
SMOVL C01500 +MOVJ EC01500
ARCON
SMOVL C01501 +MOVJ EC01501
SMOVL C01502 +MOVJ EC01502
SMOVL C01503 +MOVJ EC01503
SMOVL C01504 +MOVJ EC01504
SMOVL C01505 +MOVJ EC01505
SMOVL C01506 +MOVJ EC01506
ARCOF
SMOVL C01507 +MOVJ EC01507
ARCON
SMOVL C01508 +MOVJ EC01508
SMOVL C01509 +MOVJ EC01509
SMOVL C01510 +MOVJ EC01510
SMOVL C01511 +MOVJ EC01511
SMOVL C01512 +MOVJ EC01512
SMOVL C01513 +MOVJ EC01513
ARCOF
SMOVL C01514 +MOVJ EC01514
ARCON
SMOVL C01515 +MOVJ EC01515
SMOVL C01516 +MOVJ EC01516
SMOVL C01517 +MOVJ EC01517
END
